# B&R Automation Studio project ABC_Pltzr (part 4)

### paiUDPService.typ - Global data types
```iecst
(********************************************************************
 * COPYRIGHT -- pai
 ********************************************************************
 * Package: paiUDPService
 * File: paiUDPService.typ
 * Author: goran
 * Created: October 12, 2011
 ********************************************************************
 * Data types of package paiUDPService
 ********************************************************************)

TYPE
	paiUdpConst_typ :
		(
		UDP_IP_ADDR_LEN := 32,
		UDP_SERVER_RXBUF_SIZE := 10000,
		UDP_CLIENT_TXBUF_SIZE := 10000
		);
	paiUdpIPAddress_typ : 	STRUCT
		digit3 : USINT;
		digit2 : USINT;
		digit1 : USINT;
		digit0 : USINT;
		text : STRING[20];
	END_STRUCT;
	paiUdpSystemConfig_typ : 	STRUCT
		magicNumber : UDINT; (*Magic number to detect permanent memory changes.*)
		udpClientMode : USINT; (*Outgoing (client) UDP mode of operation. 0-Echo (send status upon receiving command, needs only port number, used IP from received command), 1-Continues (needs host IP address and Port number)*)
		udpClientUpdateRate : USINT; (*Update rate (Hz) for the the UDP client when in mode 1;*)
		udpLocalServerPortNumber : UINT; (*UDP port number of the local UDP server.*)
		udpRemoteHostPortNumber : UINT; (*UDP port number of the remote host*)
		udpRemoteHostIpAddress : paiUdpIPAddress_typ; (*IP address of the remote UDP host*)
		updInterfaceType : UDINT; (*0-ISM native type; 1-Custom interface, type 1*)
	END_STRUCT;
	paiUdpStatistics_typ : 	STRUCT  (*UDP server statistics*)
		datagramCountTotal : UDINT; (*total number of received datagrams*)
		datagramPerSec : UDINT; (*number of received datagrams in the past second*)
		datagramPerSecMax : UDINT; (*max number of received datagrams in a second*)
		bytesTotal : UDINT; (*totral number of received bytes*)
		bytesPerSec : UDINT;
		bytesPerSecMax : UDINT;
		errorCountTotal : UDINT; (*total number of errors*)
	END_STRUCT;
	paiUdpClientInterface_typ : 	STRUCT
		iConnect : BOOL;
		iRmtIPAddr : STRING[UDP_IP_ADDR_LEN];
		iRmtUdpPort : UINT;
		iMode : USINT; (*0-echo mode (client's tx triggered by server's rx); 1-continues mode (rate timer 1 .. 100Hz used to trigger client's send) *)
		iSend : BOOL;
		iSendEcho : BOOL;
		iSendEchoRmtIpAddr : STRING[UDP_IP_ADDR_LEN];
		iUpdateRate : USINT;
		iTaskCycleTimeXms : USINT;
		iTxDataAdr : UDINT;
		iTxDataLen : UDINT;
		iTxCallback : UDINT;
		oError : BOOL;
		oRmtIpAddr : STRING[UDP_IP_ADDR_LEN];
		oRmtUdpPort : UINT;
		oConnected : BOOL;
		oSendDone : BOOL;
	END_STRUCT;
	paiUdpServerInterface_typ : 	STRUCT
		iEnable : BOOL;
		iUdpServerPort : UINT;
		iRxCallback : UDINT;
		iRxTimeoutXms : UDINT;
		oRxIsTimeout : BOOL;
		oError : BOOL;
		oRxReady : BOOL;
		oRxRmtIP : STRING[UDP_IP_ADDR_LEN];
		oRxRmtPort : UINT;
		oRxDataLen : UDINT;
		oRxDataLenMax : UDINT;
		oRxDataAdr : UDINT;
	END_STRUCT;
	paiUdpFBKs_typ : 	STRUCT
		open : UdpOpen;
		close : UdpClose;
		connect : UdpConnect;
		disconnect : UdpDisconnect;
		recv : UdpRecv;
		send : UdpSend;
		ioctl : UdpIoctl;
	END_STRUCT;
	paiUdpClient_typ : 	STRUCT
		clientIf : paiUdpClientInterface_typ;
		client : paiUdpFBKs_typ;
		txStats : paiUdpStatistics_typ;
		sm : bgSSM_typ;
		txbuf : ARRAY[0..UDP_CLIENT_TXBUF_SIZE]OF USINT;
	END_STRUCT;
	paiUdpServer_typ : 	STRUCT
		serverIf : paiUdpServerInterface_typ;
		server : paiUdpFBKs_typ;
		rxStats : paiUdpStatistics_typ;
		sm : bgSSM_typ;
		rmtIPAddr : STRING[UDP_IP_ADDR_LEN];
		rxlen : UDINT;
		rxbuf : ARRAY[0..UDP_SERVER_RXBUF_SIZE]OF USINT;
	END_STRUCT;
END_TYPE
```

### paiUDPService.var - Global variables
```iecst
(********************************************************************
 * COPYRIGHT -- pai
 ********************************************************************
 * Package: paiUDPService
 * File: paiUDPService.var
 * Author: goran
 * Created: October 12, 2011
 ********************************************************************
 * Variables of package paiUDPService
 ********************************************************************)
VAR CONSTANT
	gUdpServer_DefaultPort : UDINT := 9999; (*UDP Server default port*)
	gUdpClient_TaskCycleTimeXms : UDINT := 1; (*UDP Client task cycle time in [ms]*)
	gUdpClient_DefaultPort : UDINT := 9998; (*UDP Client default port*)
END_VAR
VAR
	gUdpClient_DefaultHostAdr : STRING[UDP_IP_ADDR_LEN] := '127.0.0.1'; (*UDP Client default host IP address when using continues UDP client mode*)
END_VAR
VAR RETAIN
	gUdpSystemCfg : paiUdpSystemConfig_typ := (0); (*UDP System Configuration Data (remanent memory)*)
END_VAR
VAR
	gUdpServer : paiUdpServer_typ; (*UDP Server Object Instance*)
	gUdpClient : paiUdpClient_typ; (*UDP Client Object Instance*)
END_VAR
```

### paiUdpserv.c - Implementation code
```c
/********************************************************************
 * COPYRIGHT -- pai
 ********************************************************************
 * Program: udpserv
 * File: udpserv.c
 * Author: goran
 * Created: October 05, 2011
 ********************************************************************
 * Implementation of program udpserv
 ********************************************************************/

#include <bur/plctypes.h>

#ifdef _DEFAULT_INCLUDES
	#include <AsDefault.h>
#endif

#include "../../libraries/sprintf2/sprintf2.h"

enum{
	udpServZero = 0,
	udpServEnable,
	udpServInit,
	udpServActive,
	udpServClose,
	udpServError,
	udpServLast
}STATEMACHINE;

static const char* udpServStateName(int state)
{
static const char* stateNames[] = {
"Zero",
"Enable",
"Init",
"Active",
"Close",
"Error",
};

	if( state >= udpServLast)
		return "unknow";

	return stateNames[state];
};

/*
###############################################################################
Utilities
###############################################################################
*/

/**
 Simple logging
 Log goes to an array of PV strings > see _LOCAL STRING log[][] variable below
 Log output is visible via Automation Studio watch window
 Example of a log statement used within the code is:
 DBG(lgr, "This is log example. %d ", value1);
 To complety disable logging from this source file, change next line to: #if 0
*/
#if 1
#include <../../bglib/bgPVLogger3.c>
#define LOG_ENTRY_COUNT 20	//max number of log entries
#define LOG_ENTRY_LENGTH  32 //max length of individual log message. Longer msg are truncated
_LOCAL STRING logUdpServ[LOG_ENTRY_COUNT][LOG_ENTRY_LENGTH]; //log output visible from Automation Studio!
#else
#define DBG(lgr, format, args...) ;
#define DBGINIT(lgr, logoutput, logEntryCount, logEntrySize)  ;
#endif

static void udpServerRxData(paiUdpServer_typ *p){
bgSSM_typ* pSm = &p->sm;

	//stats
	p->rxStats.datagramCountTotal++;
	p->rxStats.bytesTotal += p->server.recv.recvlen;

	//values for cummulative (per min) calculations
	pSm->counter[0]++;
	pSm->counter[1] +=p->server.recv.recvlen;

	//interface
	p->serverIf.oRxReady = 1;
	p->serverIf.oRxDataLen = p->server.recv.recvlen;
	p->serverIf.oRxDataAdr = (UDINT)p->rxbuf;
	p->serverIf.oRxRmtPort = p->server.recv.port;
	brsstrcpy((UDINT)p->serverIf.oRxRmtIP, (UDINT)p->rmtIPAddr);

	//execute rx callback to enable app to process received data
	if(p->serverIf.iRxCallback){
		void (*rxCallback)(UDINT pBuf, UDINT rxLen) =  ( void(*) (UDINT, UDINT) ) p->serverIf.iRxCallback;
		(*rxCallback)( (UDINT)p->rxbuf, p->server.recv.recvlen);
	}
}

/*
###############################################################################
Functions
###############################################################################
*/

static void udpServerSMCyclic(paiUdpServer_typ *p)
{
bgSSM_typ* pSm = &p->sm;

	//operate timer(s)
	bgTimerCyclic(&pSm->timer_x1ms[0]);
	bgTimerCyclic(&pSm->timer_x1ms[1]);//rx timeout timer
	bgTimerCyclic(&pSm->timer_x1ms[2]);//1 sec tick timer

	p->serverIf.oRxIsTimeout = bgTimerIsTimeOut(&pSm->timer_x1ms[1]);

	//stats timers
	if( bgTimerIsTimeOut(&pSm->timer_x1ms[2]) ){
		bgTimerStart(&pSm->timer_x1ms[2], 1000);

		//values for cummulative (per min) calculations for datagrams
		p->rxStats.datagramPerSec = pSm->counter[0];
		pSm->counter[0] = 0;
		if(p->rxStats.datagramPerSec > p->rxStats.datagramPerSecMax){
			p->rxStats.datagramPerSecMax = p->rxStats.datagramPerSec;
		}

		//values for cummulative (per min) calculations for bytes
		p->rxStats.bytesPerSec = pSm->counter[1];
		pSm->counter[1] = 0;
		if(p->rxStats.bytesPerSec > p->rxStats.bytesPerSecMax){
			p->rxStats.bytesPerSecMax = p->rxStats.bytesPerSec;
		}
	}

	/*execute control state machine cyclic handler*/
	bgSSMCyclic(pSm);
	//show change of state in a log
	if( bgSSMIsStateInit(pSm) ){
		DBG(lgr, "sm=%s(%d)", bgSSMGetStateText(pSm), bgSSMGetState(pSm));
	}

	switch(bgSSMGetState(pSm)){
		//========================================
		case udpServZero:
			bgSSMStateNext(pSm, udpServEnable);
			p->serverIf.oError = 0;
			p->serverIf.oRxReady = 0;

		break;
		//========================================
		case udpServEnable:
			if(p->serverIf.iEnable){
				bgSSMStateNext(pSm, udpServInit);
			}
		break;
		//========================================
		case udpServInit:

			if( bgSSMIsStateInit(pSm) ){

				p->server.open.enable = 1;
				p->server.open.port = p->serverIf.iUdpServerPort;
				p->server.open.pIfAddr = 0;
//IMPORTANT:
//in order for the following conditional compilation to work properly, PLC object in the Configuration view
//must contain following defintion:
//Folder: Build
//Field: Additional Build Options
//Value: -D $(AS_CONFIGURATION)
//Using the above, name of the current AS configuration (i.e. realhw1 or testsim or else) becomes
//a defined preprocessor name. As a result, it's possible to destinguish between different configurations!
//#ifdef testsim
#ifdef Simulation
				//In case of testsim (ARsim) target, don't use socket options
				p->server.open.options = 0;
#warning "Project - UDP - ARsim target!"
#else
				//For all other (real) targets, use socket options
				p->server.open.options = udpOPT_REUSEPORT;
#warning "Project - UDP - NOT an ARsim target!"
#endif
				return;
			}

			if(p->server.open.status == ERR_FUB_BUSY)
				return;

			p->server.open.enable = 0;

			if(p->server.open.status == ERR_OK){
				p->server.recv.ident = p->server.open.ident;
				p->server.send.ident = p->server.open.ident;
				p->server.close.ident = p->server.open.ident;
				p->server.connect.ident = p->server.open.ident;
				p->server.disconnect.ident = p->server.open.ident;
				p->server.ioctl.ident = p->server.open.ident;
				bgSSMStateNext(pSm, udpServActive);
				return;
			}

			DBG(lgr,"Err udp.open=%d", p->server.open.status);
			bgSSMStateNext(pSm, udpServError);

		break;
		//========================================
		case udpServActive:

			if( bgSSMIsStateInit(pSm) ){
				p->server.recv.enable = 1;

				p->server.recv.pData = (UDINT)&p->rxbuf[0];
				p->server.recv.datamax = UDP_SERVER_RXBUF_SIZE;
				p->server.recv.pIpAddr = (UDINT)&p->rmtIPAddr[0];
				p->server.recv.flags = 0;

				bgTimerStart(&pSm->timer_x1ms[1], p->serverIf.iRxTimeoutXms);

				return;
			}

			//Disabling UDP server currently not supported. Disabling (i.e. change port) requires reset
			//if(!p->serverIf.iEnable){
			//	stateNext(pSm, udpServClose);
			//}

			if((p->server.recv.status == ERR_FUB_BUSY) || (p->server.recv.status == udpERR_NO_DATA))
				return;

			p->server.recv.enable = 0;

			if(p->server.recv.status == ERR_OK){

				DBG(lgr,"udpServ rx from %s", p->rmtIPAddr);
				DBG(lgr,"rmtPort=%d, rxlen=%d", p->server.recv.port, p->server.recv.recvlen);
				udpServerRxData(p);
				return;
			}

			DBG(lgr,"Err udp.recv=%d", p->server.recv.status);
			bgSSMStateNext(pSm, udpServError);

		break;
		//========================================
		case udpServClose:

			if( bgSSMIsStateInit(pSm) ){
				DBG(lgr,"UDP Server close");
				p->server.close.enable = 1;
				p->server.recv.enable = 0;
				return;
			}

			if(p->server.close.status == ERR_FUB_BUSY)
				return;

			if(p->server.close.status){
				DBG(lgr,"Err udp.close=%d", p->server.close.status);
			}

			p->server.close.enable = 0;

			bgSSMStateNext(pSm, udpServZero);
		break;
		//========================================
		case udpServError:

			if( bgSSMIsStateInit(pSm) ){
				DBG(lgr,"UDP Server Error State");

				//start error recovery timer
				bgTimerStart(&pSm->timer_x1ms[0], 5000);
			}

			if( bgTimerIsTimeOut(&pSm->timer_x1ms[0]) ){
				//after timer exp > try to close the port and see if it recovers
				bgSSMStateNext(pSm, udpServClose);
			}

		break;
		//========================================
		default:
		break;
	}

}

static void udpServerInit(paiUdpServer_typ *p)
{
	bgSSM_typ* pSm = &p->sm;

	brsmemset((UDINT)p, 0, sizeof(paiUdpServer_typ));

	bgTimerStart(&p->sm.timer_x1ms[2], 1000);

	bgSSMInit(pSm, (UDINT)udpServStateName, 0);
}

static void udpServerCyclic(paiUdpServer_typ *p)
{
	//udp server state machine cyclic
	udpServerSMCyclic(p);

	//udp server fbk-s
	UdpOpen(&p->server.open);
	UdpClose(&p->server.close);
	UdpConnect(&p->server.connect);
	UdpDisconnect(&p->server.disconnect);
	UdpSend(&p->server.send);
	UdpRecv(&p->server.recv);
	UdpIoctl(&p->server.ioctl);

}

/*
###############################################################################
Main entry: Init & Cyclic Functions
###############################################################################
*/
void paiUdpServerInit(paiUdpServer_typ *p)
{
	/* TODO: Add code here */

	//init logger object
	DBGINIT(lgr, logUdpServ, LOG_ENTRY_COUNT, LOG_ENTRY_LENGTH);
	DBG(lgr, "INIT: paiUdpServerInit");

	//udp server init
	udpServerInit(p);

}

void paiUdpServerCyclic(paiUdpServer_typ *p)
{
	/* TODO: Add code here */
	//udp server cyclic
	udpServerCyclic(p);
}
```

### paiUdpclient.c - Implementation code
```c
/********************************************************************
 * COPYRIGHT -- pai
 ********************************************************************
 * Program: udpclient
 * File: udpclient.c
 * Author: goran
 * Created: January 23, 2013
 ********************************************************************
 * Implementation of program udpclient
 ********************************************************************/

#include <bur/plctypes.h>

#ifdef _DEFAULT_INCLUDES
	#include <AsDefault.h>
#endif

#include <../../bglib/bgstring.h>
#include "../../libraries/sprintf2/sprintf2.h"

enum{
	udpCliZero = 0,
	udpCliInit,
	udpCliOpen,
	udpCliConnect,
	udpCliIdle,
	udpCliTxData,
	udpCliDisconnect,
	udpCliClose,
	udpCliError,
	udpCliLast
}STATEMACHINE;

static const char* udpCliStateName(int state)
{
static const char* stateNames[] = {
"Zero",
"Init",
"Open",
"Connect",
"Idle",
"TxData",
"Disconnect",
"Close",
"Error",
};

	if( state >= udpCliLast)
		return "unknow";

	return stateNames[state];
};

/*
###############################################################################
Utilities
###############################################################################
*/

static void convertIPTextToDigits(paiUdpIPAddress_typ* p)
{
unsigned char txtbuffer[64];
bgStringList_typ list;

	brsstrcpy((UDINT)txtbuffer, (UDINT)(p->text));
	list.src = txtbuffer;

	bgStringSplitLine(&list, '.');
	if(list.itemCount != 4){
		p->digit3 = 0;
		p->digit2 = 0;
		p->digit1 = 0;
		p->digit0 = 0;
		return;
	}
	p->digit3 = (USINT)brsatoi((UDINT)list.items[0]);
	p->digit2 = (USINT)brsatoi((UDINT)list.items[1]);
	p->digit1 = (USINT)brsatoi((UDINT)list.items[2]);
	p->digit0 = (USINT)brsatoi((UDINT)list.items[3]);
}

/**
 Simple logging
 Log goes to an array of PV strings > see _LOCAL STRING log[][] variable below
 Log output is visible via Automation Studio watch window
 Example of a log statement used within the code is:
 DBG(lgr, "This is log example. %d ", value1);
 To complety disable logging from this source file, change next line to: #if 0
*/
#if 1
#include <../../bglib/bgPVLogger3.c>
#define LOG_ENTRY_COUNT 20	//max number of log entries
#define LOG_ENTRY_LENGTH  32 //max length of individual log message. Longer msg are truncated
_LOCAL STRING logUdpClient[LOG_ENTRY_COUNT][LOG_ENTRY_LENGTH]; //log output visible from Automation Studio!
#else
#define DBG(lgr, format, args...) ;
#define DBGINIT(lgr, logoutput, logEntryCount, logEntrySize)  ;
#endif

/*
###############################################################################
Functions
###############################################################################
*/

static void udpClientSMCyclic(paiUdpClient_typ *p)
{
bgSSM_typ* pSm = &p->sm;

	//operate timer(s)
	bgTimerCyclic(&pSm->timer_x1ms[0]); // delay timer

	//TimerExecute(&pSm->timer2x1ms); // update rate timer (in continues mode)
	//IMPORANT: for high speed, can't use TON block > rather, use cycle time
	if(pSm->timer_x1ms[1].ET)
		pSm->timer_x1ms[1].ET--;

	bgTimerCyclic(&pSm->timer_x1ms[2]); // 1sec stats timer

	//stats timers
	if( bgTimerIsTimeOut(&pSm->timer_x1ms[2]) ){
		bgTimerStart(&pSm->timer_x1ms[2], 1000);

		//values for cummulative (per min) calculations for datagrams
		p->txStats.datagramPerSec = pSm->counter[0];
		pSm->counter[0] = 0;
		if(p->txStats.datagramPerSec > p->txStats.datagramPerSecMax){
			p->txStats.datagramPerSecMax = p->txStats.datagramPerSec;
		}

		//values for cummulative (per min) calculations for bytes
		p->txStats.bytesPerSec = pSm->counter[1];
		pSm->counter[1] = 0;
		if(p->txStats.bytesPerSec > p->txStats.bytesPerSecMax){
			p->txStats.bytesPerSecMax = p->txStats.bytesPerSec;
		}
	}

	/*execute control state machine cyclic handler*/
	bgSSMCyclic(pSm);

	//show change of state in a log
	if( bgSSMIsStateInit(pSm) ){
		DBG(lgr, "sm=%s(%d)", bgSSMGetStateText(pSm), bgSSMGetState(pSm));
	}

	switch( bgSSMGetState(pSm) ){
		//========================================
		case udpCliZero:
			bgSSMStateNext(pSm, udpCliInit);
		break;
		//========================================
		case udpCliInit:
			if(p->clientIf.iConnect){
				bgSSMStateNext(pSm, udpCliOpen);
			}
		break;
		//========================================
		case udpCliOpen:

			if( bgSSMIsStateInit(pSm) ){
				p->client.open.enable = 1;
				p->client.open.port = 0;
				p->client.open.pIfAddr = 0;
//IMPORTANT:
//in order for the following conditional compilation to work properly, PLC object in the Configuration view
//must contain following defintion:
//Folder: Build
//Field: Additional Build Options
//Value: -D $(AS_CONFIGURATION)
//Using the above, name of the current AS configuration (i.e. realhw1 or testsim or else) becomes
//a defined preprocessor name. As a result, it's possible to destinguish between different configurations!
//#ifdef testsim
#ifdef Simulation
				//In case of testsim (ARsim) target, don't use socket options
				p->client.open.options = 0;
#warning "UDP Client - ARsim target!"
#else
				//For all other (real) targets, use socket options
				p->client.open.options = udpOPT_REUSEPORT | udpOPT_BROADCAST;
#warning "UDP Client - real target!"
#endif
				return;
			}

			if(p->client.open.status == ERR_FUB_BUSY)
				return;

			p->client.open.enable = 0;

			if(p->client.open.status == ERR_OK){
				p->client.recv.ident = p->client.open.ident;
				p->client.send.ident = p->client.open.ident;
				p->client.close.ident = p->client.open.ident;
				p->client.connect.ident = p->client.open.ident;
				p->client.disconnect.ident = p->client.open.ident;
				p->client.ioctl.ident = p->client.open.ident;
				bgSSMStateNext(pSm, udpCliConnect);
				return;
			}

			DBG(lgr,"Err udp.open=%d", p->client.open.status);
			bgSSMStateNext(pSm, udpCliError);

		break;
		//========================================
		case udpCliConnect:

			if( bgSSMIsStateInit(pSm) ){
				p->client.connect.enable = 1;
				p->client.connect.port = p->clientIf.iRmtUdpPort;
				p->client.connect.pHost = (UDINT)p->clientIf.iRmtIPAddr;
				return;
			}

			if(p->client.connect.status == ERR_FUB_BUSY)
				return;

			//p->client.connect.enable = 0;

			if(p->client.connect.status == ERR_OK){
				brsstrcpy((UDINT)p->clientIf.oRmtIpAddr, (UDINT)p->clientIf.iRmtIPAddr);
				p->clientIf.oRmtUdpPort = p->clientIf.iRmtUdpPort;

				bgSSMStateNext(pSm, udpCliIdle);
				return;
			}

			DBG(lgr,"Err udp.connect=%d", p->client.connect.status);
			bgSSMStateNext(pSm, udpCliError);

		break;
		//========================================
		case udpCliIdle:

			if( bgSSMIsStateInit(pSm) ){

			}

			//udp client in echo mode!?
			//check for iSendEcho set by the server upon it receives a message > client sends out to the same host
			if(!p->clientIf.iMode && p->clientIf.iSendEcho){
				p->clientIf.iSendEcho = 0;
				p->clientIf.iSend = 1;
				brsstrcpy((UDINT)p->clientIf.iRmtIPAddr, (UDINT)p->clientIf.iSendEchoRmtIpAddr);
			}

			//udp client in continues mode!?
			//trigger send update at a configured rate to a defined (sipplied to the inputs) remote host/port
			if(p->clientIf.iMode){

				if(!pSm->timer_x1ms[1].ET){
					int updateTimeMs;

					if( p->clientIf.iUpdateRate ){
						updateTimeMs = 1000 /  p->clientIf.iUpdateRate;
					}else{
						updateTimeMs = 1000;
					}

					if(updateTimeMs < 10)
						updateTimeMs = 12;

					if(updateTimeMs > 1000)
						updateTimeMs = 1000;

					if(p->clientIf.iTaskCycleTimeXms){
						pSm->timer_x1ms[1].ET= updateTimeMs / p->clientIf.iTaskCycleTimeXms;
					}else{
						pSm->timer_x1ms[1].ET= updateTimeMs / gUdpClient_TaskCycleTimeXms; // devide by task clas time to find out increments
					}

					p->clientIf.iSend = 1;
				}

			}

			//monitor for change in remote host settings
			//in case of a change > reconnect (disconncet then connect)
			if((p->clientIf.oRmtUdpPort != p->clientIf.iRmtUdpPort) ||
				brsstrcmp((UDINT)p->clientIf.oRmtIpAddr, (UDINT)p->clientIf.iRmtIPAddr)
			){
				DBG(lgr,"rmt settings changed. Triggering reconnect.");
				bgSSMStateNext(pSm, udpCliDisconnect);
				return;
			}

			//monitor request to send
			if(p->clientIf.iSend){
				p->clientIf.iSend = 0;

				if(p->clientIf.iTxDataLen > UDP_CLIENT_TXBUF_SIZE){
					p->clientIf.iTxDataLen = UDP_CLIENT_TXBUF_SIZE;
				}

				if(!p->clientIf.iTxDataAdr && !p->clientIf.iTxCallback){
					DBG(lgr,"udp.send nothing to tx");
					return;
				}

				//execute memcpy if datasource is defined
				if(p->clientIf.iTxDataAdr){
					brsmemcpy((UDINT)(p->txbuf), (UDINT)(p->clientIf.iTxDataAdr), p->clientIf.iTxDataLen);
				}

				//execute callback to enable app to populate data before sending
				//NOTE: callback will overwrite effect of the above memcpy if both a defined!!!
				if(p->clientIf.iTxCallback){
					void (*txCallback)(UDINT pBuf, UDINT lenTxBuf, UDINT* pLenData) =  ( void(*) (UDINT, UDINT, UDINT*) ) p->clientIf.iTxCallback;
					(*txCallback)( (UDINT)&p->txbuf[0], UDP_CLIENT_TXBUF_SIZE, &p->clientIf.iTxDataLen);
				}

				p->client.send.enable = 1;
				p->client.send.pData = (UDINT)&p->txbuf[0];
				p->client.send.datalen = p->clientIf.iTxDataLen;

				//stats
				p->txStats.datagramCountTotal++;
				p->txStats.bytesTotal += p->client.send.datalen;

				//values for cummulative (per min) calculations
				pSm->counter[0]++;
				pSm->counter[1] +=p->client.send.datalen;

				bgSSMStateNext(pSm, udpCliTxData);
				return;
			}

		break;
		//========================================
		case udpCliTxData:
			if( bgSSMIsStateInit(pSm) ){

			}

			if(p->client.send.status == ERR_FUB_BUSY)
				return;

			p->client.send.enable = 0;

			if(p->client.send.status == ERR_OK){
				p->clientIf.oSendDone = 1;
				DBG(lgr,"udp.send OK");
				bgSSMStateNext(pSm, udpCliIdle);
				return;
			}

			DBG(lgr,"Err udp.send=%d", p->client.send.status);
			bgSSMStateNext(pSm, udpCliError);

		break;
		//========================================
		case udpCliDisconnect:

			if( bgSSMIsStateInit(pSm) ){
				p->client.connect.enable = 0;
				p->client.disconnect.enable = 1;
				return;
			}

			if(p->client.disconnect.status == ERR_FUB_BUSY)
				return;

			p->client.disconnect.enable = 0;

			if(p->client.disconnect.status == ERR_OK){
				bgSSMStateNext(pSm, udpCliClose);
				return;
			}

			DBG(lgr,"Err udp.disconnect=%d", p->client.disconnect.status);
			bgSSMStateNext(pSm, udpCliClose);

		break;
		//========================================
		case udpCliClose:

			if( bgSSMIsStateInit(pSm) ){
				DBG(lgr,"UDP Client close");
				p->client.close.enable = 1;
				return;
			}

			if(p->client.close.status == ERR_FUB_BUSY)
				return;

			if(p->client.close.status){
				DBG(lgr,"Err udp.close=%d", p->client.close.status);
			}

			p->client.close.enable = 0;

			bgSSMStateNext(pSm, udpCliZero);
		break;
		//========================================
		case udpCliError:

			if( bgSSMIsStateInit(pSm) ){
				DBG(lgr,"UDP Client Error State");

				//start error recovery timer
				bgTimerStart(&pSm->timer_x1ms[0], 5000);
			}

			if( bgTimerIsTimeOut(&pSm->timer_x1ms[0]) ){
				//after timer exp > try to close the port and see if it recovers
				bgSSMStateNext(pSm, udpCliDisconnect);
			}

		break;
		//========================================
		default:
		break;
	}

}

void udpClientInit(paiUdpClient_typ *p)
{
	bgSSM_typ* pSm = &p->sm;

	bgTimerStart(&p->sm.timer_x1ms[2], 1000);

	bgSSMInit(pSm, (UDINT)udpCliStateName, 0);

}

void udpClientCyclic(paiUdpClient_typ *p)
{

	//udp client state machine
	udpClientSMCyclic(p);

	//udp client fbk-s
	UdpOpen(&p->client.open);
	UdpClose(&p->client.close);
	UdpConnect(&p->client.connect);
	UdpDisconnect(&p->client.disconnect);
	UdpSend(&p->client.send);
	UdpRecv(&p->client.recv);
	UdpIoctl(&p->client.ioctl);
}
/*
###############################################################################
Main entry: Init & Cyclic Functions
###############################################################################
*/

void paiUdpClientInit(paiUdpClient_typ *p)
{
	/* TODO: Add code here */

	//init logger object
	DBGINIT(lgr, logUdpClient, LOG_ENTRY_COUNT, LOG_ENTRY_LENGTH);
	DBG(lgr, "INIT: paiUdpClientInit");

	udpClientInit(p);

	//upd client application specific init
	p->clientIf.iConnect = 1;
#if 0

	//RESTORE SETTINGS FROM THE REMANENT STORAGE
	//sanity check for remote host ip address
	convertIPTextToDigits(&gUdpSystemCfg.udpRemoteHostIpAddress);

	if(!gUdpSystemCfg.udpRemoteHostIpAddress.digit0 ||
		!gUdpSystemCfg.udpRemoteHostIpAddress.digit1 ||
		!gUdpSystemCfg.udpRemoteHostIpAddress.digit2 ||
		!gUdpSystemCfg.udpRemoteHostIpAddress.digit3
	){
		brsstrcpy((UDINT)gUdpSystemCfg.udpRemoteHostIpAddress.text, (UDINT)gUdpClient_DefaultHostAdr);
		convertIPTextToDigits(&gUdpSystemCfg.udpRemoteHostIpAddress);
	}
	brsstrcpy((UDINT)gUdpClient.clientIf.iRmtIPAddr, (UDINT)gUdpSystemCfg.udpRemoteHostIpAddress.text);

	//sanity check for remote host UDP port number
	if(!gUdpSystemCfg.udpRemoteHostPortNumber){
		gUdpSystemCfg.udpRemoteHostPortNumber = gUdpClient_DefaultPort;
	}
	gUdpClient.clientIf.iRmtUdpPort = gUdpSystemCfg.udpRemoteHostPortNumber;

	// udpClientMode
	// 0-echo mode (send status after receiving a command from the host. Uses received IP address and UDP port number configured here.
	// 1-continues mode (send status independantly to configured 	remoteIpAddress. remoteUDP port at the configure UDP rate
	if(gUdpSystemCfg.udpClientMode > 1){
		gUdpSystemCfg.udpClientMode = 0;
	}
	gUdpClient.clientIf.iMode = gUdpSystemCfg.udpClientMode;

	// udpClientUpdateRate
	// rate to send outgoing status to remote host in case of UDP client mode 1
	//
	if(gUdpSystemCfg.udpClientUpdateRate < 1){
		gUdpSystemCfg.udpClientUpdateRate  = 1;
	}
	if(gUdpSystemCfg.udpClientUpdateRate > 100){
		gUdpSystemCfg.udpClientUpdateRate  = 100;
	}
	gUdpClient.clientIf.iUpdateRate = gUdpSystemCfg.udpClientUpdateRate;

	gUdpClient.clientIf.iSend = 0;

#endif
	//dgsUdpClientInit();
}

void  paiUdpClientCyclic(paiUdpClient_typ *p)
{
	/* TODO: Add code here */

	//udp client cyclic
	udpClientCyclic(p);

#if 0
	//in continues client mode, use localy configured settings!
	if(/*gUdpSystemCfg.udpClientMode &&*/
		((gUdpSystemCfg.udpClientMode != gUdpClient.clientIf.iMode) ||
		(gUdpClient.clientIf.iUpdateRate != gUdpSystemCfg.udpClientUpdateRate) ||
		brsstrcmp((UDINT)gUdpClient.clientIf.iRmtIPAddr, (UDINT)gUdpSystemCfg.udpRemoteHostIpAddress.text))
	){
		gUdpClient.clientIf.iMode = gUdpSystemCfg.udpClientMode;
		gUdpClient.clientIf.iUpdateRate = gUdpSystemCfg.udpClientUpdateRate;
 		brsstrcpy((UDINT)gUdpClient.clientIf.iRmtIPAddr, (UDINT)gUdpSystemCfg.udpRemoteHostIpAddress.text);
	}

	//in echo mode, just monitor for iMode change
	if(!gUdpSystemCfg.udpClientMode &&
		((gUdpSystemCfg.udpClientMode != gUdpClient.clientIf.iMode) )
	){
		gUdpClient.clientIf.iMode = gUdpSystemCfg.udpClientMode;
	}

	//in both modes use configured port number for the remote UDP host
	gUdpClient.clientIf.iRmtUdpPort = gUdpSystemCfg.udpRemoteHostPortNumber;

	//udp client cyclic
	//dgsUdpClientCyclic();
#endif
}
```

### paiUdpService.h
```c
/********************************************************************
 * COPYRIGHT --
 ********************************************************************
 * Package: paiUDPService
 * File: paiUdpService.h
 * Author: goran
 * Created: June 22, 2015
 *******************************************************************/

#include <bur/plctypes.h>

#ifdef _DEFAULT_INCLUDES
	#include <AsDefault.h>
#endif

void paiUdpServerInit(paiUdpServer_typ *p);
void paiUdpServerCyclic(paiUdpServer_typ *p);
void paiUdpClientInit(paiUdpClient_typ *p);
void paiUdpClientCyclic(paiUdpClient_typ *p);
```

### Program Logical/paiComponents/paiUDP/udpApp

#### udpApp.c
```c
/********************************************************************
 * COPYRIGHT -- pai
 ********************************************************************
 * Program: appUDP
 * File: appUDP.c
 * Author: goran
 * Created: Jan 25, 2013
 ********************************************************************
 * Implementation of program appUDP
 ********************************************************************/

#include <bur/plctypes.h>

#ifdef _DEFAULT_INCLUDES
	#include <AsDefault.h>
#endif

#include <../../../libraries/sscanf2/sscanf2.h>
#include <../paiUdpService/paiUdpService.h>
#include "../../libraries/sprintf2/sprintf2.h"
#include "../../libraries/bgringbuf/bgringbuffer.h"

#include <../../../ProjGlob/ipc.h>
#include "../../../ProjGlob/GlobalDec.h"

/*
###############################################################################
Utilities
###############################################################################
*/

/**
 Simple logging
 Log goes to an array of PV strings > see _LOCAL STRING log[][] variable below
 Log output is visible via Automation Studio watch window
 Example of a log statement used within the code is:
 DBG(lgr, "This is log example. %d ", value1);
 To complety disable logging from this source file, change next line to: #if 0
IMPORTANT:
==========
DBGINIT() statement MUST BE PLACED as a first statement within the task _INIT function!
Example:
void _INIT myTaskINIT(void)
{
	//TODO: Add code here
	//init logger object
	DBGINIT(lgr, log, LOG_ENTRY_COUNT, LOG_ENTRY_LENGTH);
}
*/
#if 1
#include <../../bglib/bgPVLogger3.c>
#define LOG_ENTRY_COUNT 100	//max number of log entries
#define LOG_ENTRY_LENGTH  100 //max length of individual log message. Longer msg are truncated
_LOCAL STRING logUdpApp[LOG_ENTRY_COUNT][LOG_ENTRY_LENGTH]; //log output visible from Automation Studio!
#else
#define DBG(lgr, format, args...) ;
#define DBGINIT(lgr, logoutput, logEntryCount, logEntrySize)  ;
#endif

/**
###############################################################################
UDP Server Receive function
###############################################################################
*/
static void udpServerCallback(UDINT pRxBuffer, UDINT lenRxData)
{

	DBG(lgr, "udpServerCallback lenRxData=%d\n\r", lenRxData);
}

/**
###############################################################################
UDP callback functions
###############################################################################
*/
//UDP Server Receive function
static void udpServerCallbackAfterReceive(UDINT pRxBuffer, UDINT lenRxData)
{
	udpServerCallback(pRxBuffer, lenRxData);
}

//UDP Client Send Callback function
static void udpClientCallback(UDINT pTxBuffer, UDINT lenTxBuffer, UDINT* pTxDataLen)
{
//	(*pTxDataLen) = brsstrlen((UDINT)&gUdpClient.txbuf[0]);
}

//UDP Client Send Callback function
static void udpClientCallbackBeforeSend(UDINT pTxBuffer, UDINT lenTxBuffer, UDINT* pTxDataLen)
{
	udpClientCallback(pTxBuffer, lenTxBuffer, pTxDataLen);
}

/*
###############################################################################
UDP communication timeout handler
###############################################################################
*/
static void	udpTimeOutHandler()
{
	//application logic - an example of handling a UDP receive timeout event
	//static BOOL oldRxTimeout;
	if( gUdpRxState && bgTimerIsTimeOut(&gUdpCommTimeoutTmr) /*&& !gYPAlarms.alarmActive[APP_ALARM_DBPROXYTIMEOUT]*/){
		DBG(lgr, "udp server rx timeout");
		//gYPAlarms.alarmActive[APP_ALARM_DBPROXYTIMEOUT] = gConfig.active.diag.disableDBProxTimeoutAlarm ? 0 : 1;
	}
}

/*
###############################################################################
Task execution entry points: Init & Cyclic Functions
###############################################################################
*/
void _INIT udpAppINIT(void)
{

	/* TODO: Add code here */
	//init logger object
	DBGINIT(lgr, logUdpApp, LOG_ENTRY_COUNT, LOG_ENTRY_LENGTH);
	DBG(lgr, "INIT: udpAppINIT");

	//Init UDP server object
	//======================
	paiUdpServerInit(&gUdpServer);
	//Set UDP server related parameters
	//Define application specific UDP server rx callback function
	gUdpServer.serverIf.iRxCallback = (UDINT)udpServerCallbackAfterReceive;
	gUdpServer.serverIf.oRxDataLenMax = UDP_SERVER_RXBUF_SIZE;
	gUdpServer.serverIf.iEnable = 1;
	gUdpServer.serverIf.iUdpServerPort = 9999;

	//Init UDP client object
	//======================
	paiUdpClientInit(&gUdpClient);

	//Define application specific UDP client tx callback function
	gUdpClient.clientIf.iTxCallback = (UDINT)udpClientCallbackBeforeSend;

	//Adjust UDP client/server settings according to the application needs (i.e. use HMI if needed)
	//For other defaults see:
	//paiUDPService.var (i.e. defined UDP related const)
	//udpserv.c/udpservINIT() and udpclient.c/udpclientINIT()
	gUdpSystemCfg.udpClientMode = 0;//not continues mode
	gUdpSystemCfg.udpClientUpdateRate = 10;//[Hz]
	//strcpy(gUdpSystemCfg.udpRemoteHostIpAddress.text, "192.168.100.31");
	//strcpy(gUdpSystemCfg.udpRemoteHostIpAddress.text, "192.168.100.171");
	brsstrcpy((UDINT)gUdpSystemCfg.udpRemoteHostIpAddress.text, (UDINT)"192.168.100.255");
	//strcpy(gUdpSystemCfg.udpRemoteHostIpAddress.text, "192.168.100.10");
	//strcpy(gUdpSystemCfg.udpRemoteHostIpAddress.text, "127.0.0.1");
	//strcpy(gUdpSystemCfg.udpRemoteHostIpAddress.text, "192.168.100.255");
	gUdpClient.clientIf.iTaskCycleTimeXms = 1;//udp client runs under 10ms cycle time
	gUdpServer.serverIf.iRxTimeoutXms = 4000;//udp server rx timeout time

	//bgTimerStart(&gUdpCommTimeoutTmr, gConfig.active.hmi.dbProxyCommTimeout * 1000.0);//start response timeout timer
	bgTimerStart(&gUdpCommTimeoutTmr, 5000);//start response timeout timer

}

//typedef union TAppIpcMsgXXX
//{
//    UDINT gen;
//    USINT rw_shm;
//    DINT  errMsg;
//}TAppIpcMsgXXX_typ;
//

void _CYCLIC udpAppCYCLIC(void)
{
	/* TODO: Add code here */

	//operate timer
	bgTimerCyclic(&gUdpCommTimeoutTmr) ;

	//application logic - on send complete, copy status into last statusSent
	if(gUdpClient.clientIf.oSendDone){
		gUdpClient.clientIf.oSendDone = 0;

		overheadIpcUDPTxClientCyclic( &gIpcCommFifoMem );

		//preset response timeout timer
//		gUdpRxState = 1; //need to receive a response
		if( bgTimerIsTimeOut(&gUdpCommTimeoutTmr) ){
			//bgTimerStart(&gUdpCommTimeoutTmr, gConfig.active.hmi.dbProxyCommTimeout * 1000.0);//start response timeout timer
			bgTimerStart(&gUdpCommTimeoutTmr, 5000);//start response timeout timer
		}
	}

	//application logic - en example of handling a UDP rx event
	if(gUdpServer.serverIf.oRxReady){
		//gUdpServer.serverIf.oRxReady = 0; //Consumer of the message shall clear this bit
		gUdpRxState = 0; //response received
		//gYPAlarms.alarmActive[APP_ALARM_DBPROXYTIMEOUT] = 0;//clear DB proxy alarm
	}

	//handle a UDP rx timeout
	udpTimeOutHandler();

	//cyclic execution of the UDP related services
	paiUdpServerCyclic(&gUdpServer);
	paiUdpClientCyclic(&gUdpClient);
}
//EOF
```

### paiUser.typ - pai Mp types
```iecst
(********************************************************************
 * COPYRIGHT -- pai
 ********************************************************************
 * Package: paiTemplate
 * File: paiUser.typ
 * Author: goran
 * Created: August 28, 2013
 ********************************************************************
 * Data types of package paiUser
 ********************************************************************)
(*########################################################################*)
(*pai specific defines for user access logic*)
(*########################################################################*)

TYPE
	paiUserAccessMaxEnums :
		(
		paiUSER_RIGHTSMAXIDX := 19, (*Access rights max index*)
		paiUSER_USERSMAXIDX := 9, (*Users max index*)
		paiUSER_GROUPMAXIDX := 5 (*Groups max index*)
		);
	paiUserAccessRightsIndex :
		(
		paiUSER_ACCESS_MFG := 0, (*Access right index*)
		paiUSER_ACCESS_ADMIN := 1, (*Access right index*)
		paiUSER_ACCESS_MAINT := 2, (*Access right index*)
		paiUSER_ACCESS_NONE := 3 (*Access right index*)
		);
	paiMpUserAccessRightEnum :
		(
		mpUSER_ACCESS_UNDEFINED := 0, (*Access right undefined*)
		mpUSER_ACCESS_NONE := 1, (*No access rights*)
		mpUSER_ACCESS_VIEW := 2, (*Read access*)
		mpUSER_ACCESS_ACTUATE := 3, (*Processes can be started/stopped but not edited*)
		mpUSER_ACCESS_FULL := 4 (*Full access (read-write access)*)
		);
	paiMpUserMgrUIGroupInfoType : 	STRUCT
		Name : STRING[20]; (*Name of the user group*)
		Index : UINT; (*Index of the user group*)
		Level : DINT; (*Level of the user group*)
		Admin : BOOL; (*Indicates whether this group has administrator rights*)
		AccessRights : ARRAY[0..19]OF paiMpUserAccessRightEnum; (*List with the access rights for individual actions*)
	END_STRUCT;
	paiUserInfo_typ : 	STRUCT
		UserName : STRING[20];
		UserFullName : STRING[100];
		Password : STRING[20];
		PIN : UDINT;
		GroupIndex : UDINT;
	END_STRUCT;
	paiUserMgrUIConnect_typ : 	STRUCT
		groupIndex : UDINT;
		groupIndexMax : UDINT;
		userIndex : UDINT;
		userIndexMax : UDINT;
		loggedIndex : UDINT;
		isUserLogged : UDINT;
		visibleLogged : UDINT;
		visibleNotLogged : UDINT;
		btnRestartLoginTimer : UDINT;
		btnToggleLogin : UDINT;
		remainingLoginTime_min : UDINT;
		remainingLoginTime_sec : UDINT;
		pwdLevel : UDINT;
		pwdLevelOld : UDINT;
		pwdLevelCompletion : UDINT;
		listUserNames : ARRAY[0..11]OF STRING[20];
		listUserPasswords : ARRAY[0..11]OF STRING[20];
	END_STRUCT;
	paiUserMgrPrivate_typ : 	STRUCT
		UIConnect : paiUserMgrUIConnect_typ;
		loginTimer : TON;
	END_STRUCT;
	paiUserConfiguration_typ : 	STRUCT
		listGroups : ARRAY[0..5]OF paiMpUserMgrUIGroupInfoType; (*table colum: id-s*)
		listUsers : ARRAY[0..9]OF paiUserInfo_typ;
		loginTime_sec : REAL;
		New_Member : USINT;
	END_STRUCT;
	paiUserMgr_typ : 	STRUCT
		currentGroup : paiMpUserMgrUIGroupInfoType;
		currentUser : paiUserInfo_typ;
		pUserConfig : REFERENCE TO paiUserConfiguration_typ;
		userMgr : paiUserMgrPrivate_typ;
	END_STRUCT;
END_TYPE
```

### paiUser.var - Global variables
```iecst
(********************************************************************
 * COPYRIGHT -- pai
 ********************************************************************
 * Package: HMI
 * File: HMI.var
 * Author: goran
 * Created: August 28, 2013
 ********************************************************************
 * Variables of package HMI
 ********************************************************************)
VAR
	gPaiUserConfig : paiUserConfiguration_typ := (0);
	gPaiUserMgr : paiUserMgr_typ := (0);
END_VAR
```

### Program Logical/paiComponents/paiUser/paiUser (ANSIC) - pai User Service (TK#8)

#### paiUser.c - Cyclic code
```c
#include <bur/plctypes.h>

#ifdef _DEFAULT_INCLUDES
	#include <AsDefault.h>
#endif

/*
###############################################################################
PAI_CONFIGURATION_SECTION
Code below allows configuration for:
User access
###############################################################################
*/
#warning "pai Configuration: User Access"

//=============================================================================
//User Login support
//=============================================================================
static void paiUserInitGroups()
{
	int ii;
	int groupIndex;

	gPaiUserConfig.loginTime_sec = 60.0 * 30.0;//30 minutes

	groupIndex = 0;
	brsstrcpy((UDINT)gPaiUserConfig.listGroups[groupIndex].Name, (UDINT)"NotLogged");
	gPaiUserConfig.listGroups[groupIndex].Level = 0;
	gPaiUserConfig.listGroups[groupIndex].Admin = 0;
	for(ii=0; ii<=paiUSER_RIGHTSMAXIDX;ii++){
		gPaiUserConfig.listGroups[groupIndex].AccessRights[ii] = mpUSER_ACCESS_UNDEFINED;
	}

	groupIndex = 1;
	brsstrcpy((UDINT)gPaiUserConfig.listGroups[groupIndex].Name, (UDINT)"Operator");
	gPaiUserConfig.listGroups[groupIndex].Level = 10;
	gPaiUserConfig.listGroups[groupIndex].Admin = 0;
	for(ii=0; ii<=paiUSER_RIGHTSMAXIDX;ii++){
		gPaiUserConfig.listGroups[groupIndex].AccessRights[ii] = mpUSER_ACCESS_FULL;
	}

	groupIndex = 2;
	brsstrcpy((UDINT)gPaiUserConfig.listGroups[groupIndex].Name, (UDINT)"Maintenance");
	gPaiUserConfig.listGroups[groupIndex].Level = 20;
	gPaiUserConfig.listGroups[groupIndex].Admin = 0;
	for(ii=0; ii<=paiUSER_RIGHTSMAXIDX;ii++){
		gPaiUserConfig.listGroups[groupIndex].AccessRights[ii] = mpUSER_ACCESS_FULL;
	}

	groupIndex = 3;
	brsstrcpy((UDINT)gPaiUserConfig.listGroups[groupIndex].Name, (UDINT)"Supervisor");
	gPaiUserConfig.listGroups[groupIndex].Level = 30;
	gPaiUserConfig.listGroups[groupIndex].Admin = 0;
	for(ii=0; ii<=paiUSER_RIGHTSMAXIDX;ii++){
		gPaiUserConfig.listGroups[groupIndex].AccessRights[ii] = mpUSER_ACCESS_FULL;
	}

	groupIndex = 4;
	brsstrcpy((UDINT)gPaiUserConfig.listGroups[groupIndex].Name, (UDINT)"Manufacturer");
	gPaiUserConfig.listGroups[groupIndex].Level = 100;
	gPaiUserConfig.listGroups[groupIndex].Admin = 1;
	for(ii=0; ii<=paiUSER_RIGHTSMAXIDX;ii++){
		gPaiUserConfig.listGroups[groupIndex].AccessRights[ii] = mpUSER_ACCESS_FULL;
	}

}

static void paiUserUpdatePWDUI()
{
	int ii;

	brsstrcpy((UDINT)gPaiUserMgr.userMgr.UIConnect.listUserNames[0]  ,(UDINT)"n.a.");
	brsstrcpy((UDINT)gPaiUserMgr.userMgr.UIConnect.listUserPasswords[0], (UDINT)"not used PIN");
	for(ii = 1; ii <=(paiUSER_USERSMAXIDX+1); ii++){
		brsstrcpy((UDINT)gPaiUserMgr.userMgr.UIConnect.listUserNames[ii]  ,(UDINT)gPaiUserConfig.listUsers[ii-1].UserName);
		brsitoa((UDINT)gPaiUserConfig.listUsers[ii-1].PIN, (UDINT)gPaiUserMgr.userMgr.UIConnect.listUserPasswords[ii] );
	}

}

static void paiUserInitUsers()
{
	int userIndex;

	userIndex = 0;
	brsstrcpy((UDINT)gPaiUserConfig.listUsers[userIndex].UserName, (UDINT)"Operator");
	brsstrcpy((UDINT)gPaiUserConfig.listUsers[userIndex].UserFullName, (UDINT)"Mach. Operator");
	gPaiUserConfig.listUsers[userIndex].PIN = 24025;
	gPaiUserConfig.listUsers[userIndex].GroupIndex = 1;

	userIndex = 1;
	brsstrcpy((UDINT)gPaiUserConfig.listUsers[userIndex].UserName, (UDINT)"Maintenance");
	brsstrcpy((UDINT)gPaiUserConfig.listUsers[userIndex].UserFullName, (UDINT)"Mach. Maintenance");
	//gPaiUserConfig.listUsers[userIndex].PIN = 9375144;
	gPaiUserConfig.listUsers[userIndex].PIN = 4858418;//changed on 9/21/2016, request from customer
	gPaiUserConfig.listUsers[userIndex].GroupIndex = 2;

	userIndex = 2;
	brsstrcpy((UDINT)gPaiUserConfig.listUsers[userIndex].UserName, (UDINT)"ABC Service");
	brsstrcpy((UDINT)gPaiUserConfig.listUsers[userIndex].UserFullName, (UDINT)"ABC Pckg.");
	gPaiUserConfig.listUsers[userIndex].PIN = 81134689;
	gPaiUserConfig.listUsers[userIndex].GroupIndex = 4;

//	userIndex = 3;
//	brsstrcpy(gPaiUserConfig.listUsers[userIndex].UserName, "user4");
//	brsstrcpy(gPaiUserConfig.listUsers[userIndex].UserFullName, "User Four");
//	gPaiUserConfig.listUsers[userIndex].PIN = 4444;
//	gPaiUserConfig.listUsers[userIndex].GroupIndex = 4;

	gPaiUserMgr.userMgr.UIConnect.userIndex = 0;
	gPaiUserMgr.userMgr.UIConnect.userIndexMax = userIndex;

	paiUserUpdatePWDUI();
}

static void	paiUserMgrInit()
{
	gPaiUserMgr.pUserConfig = &gPaiUserConfig;

	gPaiUserMgr.userMgr.UIConnect.pwdLevel = 0;
	gPaiUserMgr.userMgr.UIConnect.pwdLevelOld = 0;
	gPaiUserMgr.userMgr.UIConnect.visibleNotLogged = 0;//visible
	gPaiUserMgr.userMgr.UIConnect.visibleLogged = 1;//not visible
	gPaiUserMgr.userMgr.UIConnect.loggedIndex = 0;
	gPaiUserMgr.userMgr.UIConnect.isUserLogged = 0;

	brsmemcpy((UDINT)&gPaiUserMgr.currentGroup, (UDINT)&gPaiUserConfig.listGroups[0], sizeof(gPaiUserMgr.currentGroup));
	brsmemset((UDINT)&gPaiUserMgr.currentUser, 0, sizeof(gPaiUserMgr.currentUser));
	brsstrcpy((UDINT)gPaiUserMgr.currentUser.UserName  ,(UDINT)"n.a.");
	brsstrcpy((UDINT)gPaiUserMgr.currentUser.UserFullName, (UDINT)"n.a.");

}

static void paiUserMgrCyclic()
{

	//user login activity from the login screen
	if(gPaiUserMgr.userMgr.UIConnect.pwdLevel != gPaiUserMgr.userMgr.UIConnect.pwdLevelOld){
		if(gPaiUserMgr.userMgr.UIConnect.pwdLevel == (gPaiUserMgr.userMgr.UIConnect.userIndex + 1) ){
			//user login success!
			gPaiUserMgr.userMgr.UIConnect.isUserLogged = 1;

			gPaiUserMgr.userMgr.UIConnect.loggedIndex = gPaiUserMgr.userMgr.UIConnect.userIndex;
			if(gPaiUserMgr.userMgr.UIConnect.loggedIndex > paiUSER_USERSMAXIDX){
				gPaiUserMgr.userMgr.UIConnect.loggedIndex = paiUSER_USERSMAXIDX;
			}

			gPaiUserMgr.userMgr.UIConnect.visibleNotLogged = 1;//not visible
			gPaiUserMgr.userMgr.UIConnect.visibleLogged = 0;//visible visible

			//define current user
			brsmemcpy((UDINT)&gPaiUserMgr.currentUser, (UDINT)&gPaiUserConfig.listUsers[gPaiUserMgr.userMgr.UIConnect.loggedIndex], sizeof(gPaiUserMgr.currentUser));

			//define current group
			if(gPaiUserMgr.currentUser.GroupIndex > paiUSER_GROUPMAXIDX){
				gPaiUserMgr.currentUser.GroupIndex = paiUSER_GROUPMAXIDX;
			}
			brsmemcpy((UDINT)&gPaiUserMgr.currentGroup, (UDINT)&gPaiUserConfig.listGroups[gPaiUserMgr.currentUser.GroupIndex], sizeof(gPaiUserMgr.currentGroup));

			//start timeout timer
			bgTimerStart(&gPaiUserMgr.userMgr.loginTimer, 1000 * gPaiUserMgr.pUserConfig->loginTime_sec);
		}else{
			paiUserMgrInit();
		}
	}
	gPaiUserMgr.userMgr.UIConnect.pwdLevelOld = gPaiUserMgr.userMgr.UIConnect.pwdLevel;

	//login timer expired?
	if(gPaiUserMgr.userMgr.UIConnect.isUserLogged && bgTimerIsTimeOut(&gPaiUserMgr.userMgr.loginTimer) ){
		paiUserMgrInit();
	}

	//restart login timer button pressed?
	if(gPaiUserMgr.userMgr.UIConnect.btnRestartLoginTimer){
		gPaiUserMgr.userMgr.UIConnect.btnRestartLoginTimer = 0;
		bgTimerStart(&gPaiUserMgr.userMgr.loginTimer, 1000 * gPaiUserMgr.pUserConfig->loginTime_sec);
	}

	//login button pressed?
	if(gPaiUserMgr.userMgr.UIConnect.btnToggleLogin){
		gPaiUserMgr.userMgr.UIConnect.btnToggleLogin = 0;
		if(gPaiUserMgr.userMgr.UIConnect.isUserLogged){
			paiUserMgrInit();
		}else{
			//TODO: jump to login page
			gPaiHmiMain.runtime.pageChange = 70;//login page
		}
	}

	//operate login timer
	bgTimerCyclic(&gPaiUserMgr.userMgr.loginTimer);

	//calculate remaining login time [min:sec] from remaining timer time [ms]
	gPaiUserMgr.userMgr.UIConnect.remainingLoginTime_sec = 	( bgTimerTimeRemaining(&gPaiUserMgr.userMgr.loginTimer) / 1000 ) % 60;
	gPaiUserMgr.userMgr.UIConnect.remainingLoginTime_min = 	( bgTimerTimeRemaining(&gPaiUserMgr.userMgr.loginTimer) / 1000 ) / 60;
}

//=============================================================================

void _INIT paiUserInit(void)
{
	paiUserInitGroups();
	paiUserInitUsers();
	paiUserMgrInit();

}

void _CYCLIC paiUserCyclic(void)
{
	paiUserMgrCyclic();
}
//EOF
```

### paiBnRHW.typ
```iecst
(********************************************************************
 * COPYRIGHT --
 ********************************************************************
 * Package: paiComponents
 * File: paiBRHW.typ
 * Author: goran
 * Created: June 23, 2015
 ********************************************************************
 * Data types of package paiTelnet
 ********************************************************************)

TYPE
	paiBnRHWModuleInfo_typ : 	STRUCT
		ModuleOk : BOOL;
		SerialNumber : UDINT;
		ModuleID : UINT;
		HardwareVariant : UINT;
		FirmwareVersion : UINT;
	END_STRUCT;
END_TYPE
```

### Package Logical/Globals - application types and global vars

### Messages.typ - application alarms
```iecst
(********************************************************************

 * COPYRIGHT -- Piedmont Automation Inc.

 ********************************************************************

 * File: Alarms.typ

 * Author: goran

 * Created: Jun 1, 2015

 ********************************************************************

 * Data types for project : Alarms

 ********************************************************************)

TYPE
	applicationMessages_enums :
		(
		APP_MSG_READY := 0,
		APP_MSG_RUNAUTO,
		APP_MSG_RUNDRYCYCLE,
		APP_MSG_ZEROREQUIRED,
		APS_MSG_LOWONPALLETS,
		APP_MSG_ZERO_CASETURNER,
		APP_MSG_ZERO_ROWPUSHER,
		APP_MSG_ZERO_BLADESTOP,
		APP_MSG_ZERO_TABLE,
		APP_MSG_ZERO_ELEVATOR,
		APP_MSG_ZERO_PALLETELIFT,
		APP_MSG_ZERO_RETAINERBAR,
		APP_MSG_ZERO_SQUARING,
		APP_MSG_PALLETE_COMPLETE,
		APP_MSG_DISCHARGE_BLOCKED,
		APP_MSG_STOP_BLOCK_RT,
		APP_MSG_STOP_BLOCK_LF,
		APP_MSG_PALLETE_EXITING,
		APP_MSG_ZERO_MSG18,
		APP_MSG_ZERO_MSG19,
		APP_MSG_LAST := 50
		);
END_TYPE

(*########################################################################*)
(*Application object - Message Object*)
(*########################################################################*)

TYPE
	applicationMessages_typ : 	STRUCT
		oIsMsgActive : BOOL; (*1-if alarm present*)
		msgActive : ARRAY[0..APP_MSG_LAST]OF BOOL; (*Alarms matrix. (see Visual Components Alarm System)*)
	END_STRUCT;
END_TYPE
```

### Messages.var
```iecst
(*********************************************************************************
 * Copyright: Piedmont Automation Inc
 * Author:    Goran
 * Created:   Jun 26, 2015/11:38 AM
 *********************************************************************************
 * Declaration of global variables
 *********************************************************************************)
VAR
	gMsgScroll : paiHmiMsgScrolling_typ := (0); (*Scrolling Alarm Msg Support*)
	gMessages : applicationMessages_typ := (0);
END_VAR
```

### MachineVFD.var
```iecst
(*********************************************************************************
 * Copyright: Piedmont Automation Inc
 * Author:    Goran
 * Created:   Jun 26, 2015/11:38 AM
 *********************************************************************************
 * Declaration of global variables
 *********************************************************************************)
VAR
	gMachineVFD : ARRAY[0..APP_VFD_IDXLAST] OF paiVFD_typ;
END_VAR
```

### ConfigApp.typ - Global types - machine configuration - application level - CHANGE AS NEEDED
```iecst
(********************************************************************
 * COPYRIGHT --
 ********************************************************************
 * Package: ConfigAndRecipes
 * File: appConfig.typ
 * Author: goran_2
 * Created: August 06, 2011

DEFINE APPLICATION SPECIFIC CONFIG STRUCTURES AS NEEDED

(*Insert your comment here.*)

TYPE
	appCfgEnums_typ :
		(
		New_Member
		);
	appCfgTimers_typ : 	STRUCT
		dlyTableLayerRdyToElevMove : REAL; (*delay from table layer ready before elevator moves*)
		dlyTableAtPalleteToRetBar : REAL; (*delay from table at pallete before retainter bar lowered*)
		onDlyPRRetBarDown : REAL; (*on delay for Retainer Bar Down prox switch*)
		onTmCaseTurner : REAL; (*case turner dwell time*)
		onDlyEEPallete : REAL; (*on delay for pallete/box detection PE EE2*)
		offDlyEEPallete : REAL; (*off delay for pallete/box detection PE EE2*)
		onDlyPRRetBarDown2 : REAL; (*on delay for Retainer Bar Down prox switch*)
		dlyLastCaseToRowCVStop : REAL; (*delay from Row forming complete to row push. Needed to allow box to travel.*)
		dlyRowDoneToRowPush : REAL; (*delay from Row forming complete to row push. Needed to allow box to travel.*)
		infeedCVIdleTime : REAL; (*max allowed time to run infeed cv-s before stopping them*)
		JamAlarmTmAtInfeedEE2 : REAL;
		JamAlarmTmAtRowToLongEE8 : REAL;
		JamAlarmTmRowForming : REAL;
		onDlyPalleteDischargeEE16 : REAL; (*on delay for pallete discharge sensor; longer time adjustst position of the pallete pass the sensor*)
		palletExitAlarmTm : REAL; (*pallet exit alarm time*)
		EE2OnDebounce : REAL;
		EE2OfDebounce : REAL;
		EE4OnDebounce : REAL;
		EE4OfDebounce : REAL;
		EE8OnDebounce : REAL;
		EE8OfDebounce : REAL;
		EE16OfDebounce : REAL;
		dlyPusherAtElevatorToRetract : REAL; (*dealy from pusher at extended position (et elevator) to trigger retracted motion *)
		onDlyFrontSquaring : REAL;
		onDlyTableToGrouping : REAL; (*on delay after layer is dropped onto the paller before table is moved back to grouping*)
		onDlyRetBarDown : REAL; (*On delay from the moment table starts moving to the pallet before retainer bar is lowered*)
		bladeStopOnDly1 : REAL; (*Blade stop turn on delay time; to accomoated for case traveling on the row forming belt*)
		bladeStopOnDly2 : REAL; (*Blade stop turn on delay time; to accomoated for case traveling on the row forming belt*)
		bladeStopOnDly3 : REAL; (*Blade stop turn on delay time; to accomoated for case traveling on the row forming belt*)
		bladeStopOnDly4 : REAL; (*Blade stop turn on delay time; to accomoated for case traveling on the row forming belt*)
		bladeStopOnDly5 : REAL; (*Blade stop turn on delay time; to accomoated for case traveling on the row forming belt*)
		bladeStopOnDly6 : REAL; (*Blade stop turn on delay time; to accomoated for case traveling on the row forming belt*)
	END_STRUCT;
	appCfgOptions_typ : 	STRUCT
		optTearSheetEquiped : UDINT; (*1-Tear sheet insert mechanism is present*)
		optOption1Equiped : UDINT; (*1-Tear sheet insert mechanism is present*)
		palletDispenserOption : UDINT; (*0-pallet dispenser is NOT present/NOTequipped; 1-pallet dispenser option IS present/equipped*)
		frontSquaringOption : UDINT; (*0-front squaring option is NOT present/NOTequipped; 1-front squaring option is present*)
		dryCycleCaseCount : UDINT;
		dryCycleRowCount : UDINT;
		dryCycleLayerCount : UDINT;
		tmDryCycleElevatorUp : REAL; (*time to dry cycle operation to simulate layers*)
		tmDryCycleCaseTime : REAL; (*single case loading time in dry cycle simulation*)
		dryCycleLayerDonePause : UDINT;
		tmDryCycleLayerZeroOffset : REAL; (*single case loading time in dry cycle simulation*)
	END_STRUCT;
	appCfgSystem_typ : 	STRUCT
		bladeStopCount : UDINT; (*number of blade stops (0...6)*)
		simulationMode : UDINT; (*1-yes*)
		bladeStopOnDly : ARRAY[0..APP_CFG_BLADESTOP_MAXIDX]OF REAL; (*Blade stop turn on delay time; to accomoated for case traveling on the row forming belt*)
		bladeStopDistance : ARRAY[0..APP_CFG_BLADESTOP_MAXIDX]OF REAL; (*Blade stop distance[inch]*)
		boxInfeedSide : UDINT; (*0-infeed from left to right 1-infeed from right to left; point of refernece if front of the machine infeed looking towards the table*)
	END_STRUCT;
	cfgMachineVFDs_typ : 	STRUCT
		velocitySlow_rpm : DINT; (*slow velocity (if needed)*)
		velocity_rpm : DINT; (*normal velocity*)
		acc : DINT; (*accelaration [x0.1sec]*)
		dec : DINT; (*decelaration [x0.1sec]*)
	END_STRUCT;
END_TYPE

(*######################################################*)

TYPE
	configApp_typ : 	STRUCT  (*Machine configuration includes settings for timers and settings for servo drives.*)
		system : appCfgSystem_typ;
		options : appCfgOptions_typ;
		magicNumber : UDINT;
	END_STRUCT;
END_TYPE
```

### Defaults_gConfigApp.c
```c
/********************************************************************
 * COPYRIGHT -- piedmont
 ********************************************************************
 * Program: Defaults_gConfigApp
 * File: Defaults_gConfigApp.c
 * Author: admin
 * Created: Jan 20, 2015
 ********************************************************************
 * Implementation of program Defaults_gConfigApp
 ********************************************************************/

#include <bur/plctypes.h>

#ifdef _DEFAULT_INCLUDES
 #include <AsDefault.h>
#endif

/*
###############################################################################
PAI_CONFIGURATION_SECTION
Code below allows configuration of the PV serialization / deserialization
manager.
###############################################################################
*/
#warning "app Configuration: PV Defaults for gConfigApp"

void gConfigAppDefaults()
{
int ii;

	gConfigApp.options.dryCycleCaseCount = 5;
	gConfigApp.options.dryCycleLayerCount = 3;
	gConfigApp.options.dryCycleLayerDonePause = 0;
	gConfigApp.options.palletDispenserOption = 1;
	gConfigApp.options.dryCycleRowCount = 4;
	gConfigApp.options.tmDryCycleCaseTime = 2.0;
	gConfigApp.options.tmDryCycleElevatorUp = 3.0;
	gConfigApp.options.tmDryCycleLayerZeroOffset = 2.0;

	gConfigApp.system.simulationMode = 0;
	gConfigApp.system.boxInfeedSide = 0;
	gConfigApp.system.bladeStopCount = 1;
	gConfigApp.system.bladeStopDistance[0] = 6.0;
	gConfigApp.system.bladeStopDistance[1] = 8.0;
	gConfigApp.system.bladeStopDistance[2] = 10.0;
	gConfigApp.system.bladeStopDistance[3] = 12.0;
	gConfigApp.system.bladeStopDistance[4] = 14.0;
	gConfigApp.system.bladeStopDistance[5] = 16.0;

}

void gPalletCfgDefaults()
{
	int ii;

	gPallete.palCfg.palSettings.timers.dlyTableAtPalleteToRetBar = 1.0;
	gPallete.palCfg.palSettings.timers.dlyTableLayerRdyToElevMove = 1.0;
	gPallete.palCfg.palSettings.timers.offDlyEEPallete = 1.0;
	gPallete.palCfg.palSettings.timers.onDlyPRRetBarDown = 1.0;
	gPallete.palCfg.palSettings.timers.onDlyPRRetBarDown2 = 1.0;
	gPallete.palCfg.palSettings.timers.onTmCaseTurner = 1.0;
	gPallete.palCfg.palSettings.timers.dlyRowDoneToRowPush = 1.0;
	gPallete.palCfg.palSettings.timers.dlyTableAtPalleteToRetBar = 1.0;
	gPallete.palCfg.palSettings.timers.JamAlarmTmAtInfeedEE2 = 4.0;
	gPallete.palCfg.palSettings.timers.JamAlarmTmRowForming = 4.0;
	gPallete.palCfg.palSettings.timers.JamAlarmTmAtRowToLongEE8 = 4.0;
	gPallete.palCfg.palSettings.timers.palletExitAlarmTm = 10.0;
	gPallete.palCfg.palSettings.timers.infeedCVIdleTime = 15.0;
	gPallete.palCfg.palSettings.timers.onDlyPalleteDischargeEE16 = 1.0;
	gPallete.palCfg.palSettings.timers.onDlyTableToGrouping = 0.0;
	gPallete.palCfg.palSettings.timers.EE2OfDebounce = 0.0;
	gPallete.palCfg.palSettings.timers.EE2OnDebounce = 0.0;
	gPallete.palCfg.palSettings.timers.EE4OfDebounce = 0.0;
	gPallete.palCfg.palSettings.timers.EE4OnDebounce = 0.0;
	gPallete.palCfg.palSettings.timers.EE8OfDebounce = 0.0;
	gPallete.palCfg.palSettings.timers.EE8OnDebounce = 0.0;
	gPallete.palCfg.palSettings.timers.EE16OfDebounce = 0.0;
	gPallete.palCfg.palSettings.timers.onDlyFrontSquaring = 0.0;
	gPallete.palCfg.palSettings.timers.bladeStopOnDly1 = 3.0;
	gPallete.palCfg.palSettings.timers.bladeStopOnDly2 = 3.0;
	gPallete.palCfg.palSettings.timers.bladeStopOnDly3 = 3.0;
	gPallete.palCfg.palSettings.timers.bladeStopOnDly4 = 2.0;
	gPallete.palCfg.palSettings.timers.bladeStopOnDly5 = 2.0;
	gPallete.palCfg.palSettings.timers.bladeStopOnDly6 = 2.0;

	for(ii=0; ii<=APP_VFD_IDXLAST; ii++){
		gPallete.palCfg.palSettings.vfd[ii].velocitySlow_rpm = 0.0;
		gPallete.palCfg.palSettings.vfd[ii].velocity_rpm = 0.0;
	}

	gPallete.palCfg.palSettings.vfd[1].velocitySlow_rpm = 300.0;
	gPallete.palCfg.palSettings.vfd[1].velocity_rpm = 600.0;
	gPallete.palCfg.palSettings.vfd[2].velocitySlow_rpm = 300.0;
	gPallete.palCfg.palSettings.vfd[2].velocity_rpm = 600.0;
	gPallete.palCfg.palSettings.vfd[4].velocitySlow_rpm = 300.0;
	gPallete.palCfg.palSettings.vfd[4].velocity_rpm = 600.0;
	gPallete.palCfg.palSettings.vfd[5].velocitySlow_rpm = 300.0;
	gPallete.palCfg.palSettings.vfd[5].velocity_rpm = 600.0;
	gPallete.palCfg.palSettings.vfd[6].velocitySlow_rpm = 300.0;
	gPallete.palCfg.palSettings.vfd[6].velocity_rpm = 600.0;
	gPallete.palCfg.palSettings.vfd[11].velocitySlow_rpm = 300.0;
	gPallete.palCfg.palSettings.vfd[11].velocity_rpm = 600.0;
	gPallete.palCfg.palSettings.vfd[12].velocitySlow_rpm = 300.0;
	gPallete.palCfg.palSettings.vfd[12].velocity_rpm = 600.0;

	for(ii=0; ii <= APP_VFD_IDXLAST; ii++){
		gPallete.palCfg.palSettings.vfd[ii].acc = 1;
		gPallete.palCfg.palSettings.vfd[ii].dec = 1;
	}

}
//EOF
```

### Package Logical/MachineControl - application tasks and logic

### MachineControl.typ - Global data types
```iecst
(*********************************************************************************
 * Copyright: Microsoft
 * Author:    Obed
 * Created:   May 26, 2015/11:38 AM
 *********************************************************************************
 * Declaration of AppControl global data types for ABC Palletizer
 *********************************************************************************)
(*********************************************************************************
	Application Structures
*********************************************************************************)

TYPE
	macCtrlEnums_typ :
		(
		APP_REC_MAXCASE := 12, (*Max number of cases per row*)
		APP_REC_MAXROW := 12, (*Max number of rows per layer*)
		APP_REC_MAXLAYER := 12 (*Max number of layers per palette*)
		);
END_TYPE

(*********************************************************************************
macCtrl_typ Contains all machine Control Structures. Using "mac" as abbreviation for Machine, "Ctrl" as for Control
*********************************************************************************)

TYPE
	macCtrl_typ : 	STRUCT
		main : macCtrlMain_typ; (*Machine Main*)
		infeedcv : macCtrlInfeedCV_typ; (*Timing Infeed Conveyor*)
		rowforming : macCtrlRowForming_typ; (*Row Forming Conveyor*)
		caseturner : macCtrlCaseTurner_typ; (*Case Turner*)
		retainerbar : macCtrlRetainerBar_typ;
		transfertable : macCtrlTransferTable_typ; (*Roller Transfer Table*)
		squaring : macCtrlSquaringPlates_typ; (*Main Frame Side Squaring Plates*)
		elevator : macCtrlElevator_typ; (*Main Frame Elevator*)
		palletDispenser : macCtrlPalleteDispenser_typ; (*Pallet Dispenser*)
		palletDischarge : macCtrlPalleteDischarge_typ; (*Pallet Dispenser*)
	END_STRUCT;
END_TYPE

(*********************************************************************************
macCtrlMain_typ Machine Main
*********************************************************************************)

TYPE
	macCtrlMain_typ : 	STRUCT
		modeMaintenance : BOOL; (*Mode: service/maintance. Minor or Major Fault active. Start (Auto) not possible.*)
		modeManual : BOOL; (*Mode: manual; No faults. Not in auto mode. Buttons to start auto mode IS available.*)
		modeAuto : BOOL; (*Mode: auto is active. See below for available auto modes.*)
		modeAutoProduction : BOOL; (*Mode: autoProduction; Auto. Production, Normal operation. Button to stop is available.*)
		modeAutoDryCycle : BOOL; (*Mode: autoDryCycle; Auto. DryCycleMode, Testing option. Button to stop is available.*)
		modeAutoDemo : BOOL; (*Mode: autoDemo; Auto. Demp/Show mode, Used for Show. Button to stop is available.*)
		modeAutoStarting : BOOL; (*Mode: autoStarting; Auto. Transitioning from Manual to Auto. (i.e. Start Button Pressed).*)
		modeAutoStopping : BOOL; (*Mode: autoStopping; Auto. Transitioning from Auto to Manual. (i.e. Stop Button Pressed).*)
		buttonEnabledStart : BOOL; (*Start Button control.*)
		buttonEnabledMaint : BOOL; (*Start Button control.*)
		noMajorFault : BOOL; (*No major fault on the machine.*)
		noMinorFault : BOOL; (*No minor fault on the machine.*)
		noFaults : BOOL; (*No minor or major fault on the machine.*)
		guardDoorsOk : BOOL; (*Guard door safety indicator.*)
		EStopOk : BOOL; (*EStop safety indicator.*)
		SafetyOk : BOOL; (*Safety Circuit OK*)
		VFDsNoFaults : BOOL; (*VFDs fault indication*)
		isAtZero : BOOL; (*machine is at zero position*)
		zeroIsNeeded : BOOL; (*machine is at zero position*)
		btnZero : BOOL; (*0-not pressed; 1-presed*)
		btnStart : BOOL; (*0-not pressed; 1-presed*)
		btnStop : BOOL; (*0-not pressed; 1-presed*)
		btnFaultAck : BOOL; (*1-ack fault / alarms*)
		btnClearCaseCounts : BOOL; (*1-ack fault / alarms*)
		btnZeroVisibility : INT; (*0-visible; 1-not visible*)
		hmiShowMsgZeroingNeeded : BOOL;
		btnNotInAutoModeVisibility : INT; (*0-visible; 1-not visible*)
		btnStartVisibility : INT; (*0-visible; 1-not visible*)
		btnLoadMachineCfg : BOOL;
		alwaysOnBit : BOOL; (*Always on bit*)
		testBit1 : BOOL; (*Test bit 1: TESTING ONLY! REMOVE FROM A FINAL PROGRAM!*)
		testBit2 : BOOL; (*Test bit 2: TESTING ONLY! REMOVE FROM A FINAL PROGRAM!*)
		testBit3 : BOOL; (*Test bit 3: TESTING ONLY! REMOVE FROM A FINAL PROGRAM!*)
		dummyCoil : BOOL; (*Dummy coil*)
		blink : BOOL; (*Light on/off blink signal*)
		gCamApp_btnPreview : BOOL;
		optionEStops : ARRAY[0..5]OF BOOL; (*Configuration Option for EStops Circuits*)
		optionDoorSw : ARRAY[0..5]OF BOOL; (*Configuration Options of Door Safety Switches*)
		visibleCaseInfeedOnLeft : UDINT; (*Visibility control for HMI when Case infeed on the left*)
		visibleCaseInfeedOnRight : UDINT; (*Visibility control for HMI when Case infeed on the right*)
		isDropLayerToPalletAllowed : BOOL;
		dropLayerToPalletBlock : BOOL;
		elevatorStopBlockActive : BOOL; (*Elevator stops blocks are active. This is part of the safety logic. *)
		tmrMCROnDelay : TON; (*Timer for MCR on delay*)
		tmrAirOnDelay : TON; (*Timer for air on delay*)
		tmrBlinkOn : TON; (*Timer for blink signal*)
		tmrBlinkOff : TOF; (*Timer for blink signal*)
	END_STRUCT;
END_TYPE

(*********************************************************************************
macCtrlMode_typ Machine Control Modes of Operation
*********************************************************************************)

TYPE
	macCtrlMode_typ : 	STRUCT
		Maintenance : BOOL; (*Minor or Major Fault active*)
		Manual : BOOL; (*Not in auto mode. Buttons to start auto mode are available.*)
		AutoProduction : BOOL; (*Auto. Production, Normal operation. Button to stop is available.*)
		AutoDryCycle : BOOL; (*Auto. DryCycleMode, Testing option. Button to stop is available.*)
		AutoDemo : BOOL; (*Auto. Demp/Show mode, Used for Show. Button to stop is available.*)
		AutoStarting : BOOL;
		AutoStopping : BOOL;
	END_STRUCT;
END_TYPE

(*********************************************************************************
macCtrlStats_typ Machine Statistics data (case counts, etc)
*********************************************************************************)

TYPE
	macCtrlStats_typ : 	STRUCT
		btnResetCounts : BOOL;
		btnResetCountsTotal : BOOL;
		casesPerMin : UDINT;
		caseCounter : UDINT;
		caseCounterTotal : UDINT;
		palletCounter : UDINT;
		palletCounterTotal : UDINT;
		palletTimeMin : REAL;
		palletTimeMax : REAL;
		palletTimeLast : REAL;
		runningTmr1 : TON;
		runningTmr1min : TON;
		runningTmr1sec : TON;
		palletTmr : TON;
		runTmrHours : UDINT;
		runTmrMins : UDINT;
		runTmrSec : UDINT;
		mCasesPerMinCounter : UDINT;
	END_STRUCT;
END_TYPE

(*********************************************************************************
macCtrlTimingInfeedConveyor_typ #TIMING INFEED CONVEYOR
*********************************************************************************)

TYPE
	macCtrlInfeedCV_typ : 	STRUCT
		hmiBtnOnOff : BOOL;
		infeedCvOn : BOOL;
		caseInSensorNegEdge : BOOL;
		caseInSensorPosEdge : BOOL;
		caseInSensor : BOOL;
		caseOutSensorNegEdge : BOOL;
		caseOutSensorPosEdge : BOOL;
		caseOutSensor : BOOL;
		caseAtOneCaseOnlySection : BOOL;
		nextCaseToCloseMonitorEnabled : BOOL;
		caseInfeedDone : BOOL;
		tmrJamAtCaseInSensorEE2 : TON;
		tmrJamAtCaseStageSensorEE4 : TON;
		tmrJamAtCaseOutSensorEE8 : TON;
		tmrJamRowForming : TON;
		tmrInfeedCVIdle : TON;
		tmrInfeedStopDly : TON;
		rowFormingCVRunPosEdge : BOOL;
		rowFormingCVRunNegEdge : BOOL;
		ssmInfeedCV : bgSSM_typ;
		sleepState : BOOL;
		stopRequest : BOOL;
	END_STRUCT;
END_TYPE

(*********************************************************************************
macCtrlRowFormingConveyor_typ #ROW FORMING CONVEYOR
*********************************************************************************)

TYPE
	macCtrlRowForming_typ : 	STRUCT
		isRowPusherAtHome : BOOL;
		isRowPusherAtElevator : BOOL;
		hmiBtnPusherFwdJog : BOOL;
		hmiBtnPusherRevJog : BOOL;
		hmiBtnPusherFwd : BOOL;
		hmiBtnPusherRev : BOOL;
		hmiBtnOnOffStageCV : BOOL;
		hmiBtnOnOffCV : BOOL;
		hmiBtnStopBladeUpDown1 : BOOL;
		hmiBtnStopBladeUpDown2 : BOOL;
		hmiBtnStopBladeUpDown3 : BOOL;
		hmiBtnStopBladeUpDown4 : BOOL;
		hmiBtnStopBladeUpDown5 : BOOL;
		hmiBtnStopBladeUpDown6 : BOOL;
		hmiBtnStopBladeUpDownQuick1 : BOOL;
		hmiBtnStopBladeUpDownQuick2 : BOOL;
		hmiBtnStopBladeUpDownQuick3 : BOOL;
		hmiBtnStopBladeUpDownQuick4 : BOOL;
		hmiBtnStopBladeUpDownQuick5 : BOOL;
		hmiBtnStopBladeUpDownQuick6 : BOOL;
		New_Member : USINT;
		isStopBladeUsed1 : BOOL;
		isStopBladeUsed2 : BOOL;
		isStopBladeUsed3 : BOOL;
		isStopBladeUsed4 : BOOL;
		isStopBladeUsed5 : BOOL;
		isStopBladeUsed6 : BOOL;
		allBladesDown : BOOL;
		lastCaseToStopCVDly : TON;
		rowPusherOnDly : TON;
		bladeStopOnDly : ARRAY[0..5]OF TON;
	END_STRUCT;
END_TYPE

(*********************************************************************************
macCtrlCaseTurner_typ #CASE TURNER
*********************************************************************************)

TYPE
	macCtrlCaseTurner_typ : 	STRUCT
		hmiBtnCaseTurnerUpDown : BOOL;
		hmiAutoCaseTurn : BOOL; (*0-no case turn; 1-case turn (raise turner)*)
		tmrCaseTurnerActive : TON;
	END_STRUCT;
END_TYPE

(*********************************************************************************
macCtrlRollerTransferTable_typ #ROLLER TRANSFER TABLE
*********************************************************************************)

TYPE
	macCtrlTransferTable_typ : 	STRUCT
		isTableAtGrouping : BOOL;
		isTableAtPallete : BOOL;
		hmiBtnTableFwdJog : BOOL;
		hmiBtnTableRevJog : BOOL;
		hmiBtnTableFwd : BOOL;
		hmiBtnTableRev : BOOL;
		hmiBtnOnOffCV : BOOL;
	END_STRUCT;
	macCtrlRetainerBar_typ : 	STRUCT
		revTimer : TON;
		fwdTimer : TON;
		barDwOffDlyTmr : TON;
		barDwDlyTmXms : UDINT;
		barIsUp : BOOL;
		barIsDown : BOOL;
		hmiBtnRetainterBarFwdJog : BOOL;
		hmiBtnRetainterBarRevJog : BOOL;
		hmiBtnRetainterBarFwd : BOOL;
		hmiBtnRetainterBarRev : BOOL;
	END_STRUCT;
END_TYPE

(*********************************************************************************
macCtrlElevator_typ #MAIN FRAME ELEVATOR
*********************************************************************************)

TYPE
	macCtrlElevator_typ : 	STRUCT
		elevatorIsAtTop : BOOL; (*Elevator at home position*)
		elevatorIsAboveHomeUnknown : BOOL; (*Elevator above home*)
		elevatorIsAboveNearHome : BOOL; (*Elevator above home*)
		elevatorIsAboveHome : BOOL; (*Elevator above home*)
		elevatorIsAtHome : BOOL; (*Elevator at home position*)
		elevatorIsBelowHome : BOOL; (*Elevator is below home position*)
		elevatorIsBelowNearHome : BOOL; (*Elevator is below home position*)
		elevatorIsBelowHomeUnknown : BOOL; (*Elevator is below home position, both switches out*)
		elevatorIsAtBottom : BOOL; (*Elevator at home position*)
		elevatorIsUknownPosition : BOOL; (*Elevator is below home position*)
		elevatorIsMovingUp : BOOL; (*Elevator is below home position*)
		elevatorIsMovingDw : BOOL; (*Elevator is below home position*)
		elevatorIsAtPalleteBelowHome : BOOL; (*Elevator is below home position*)
		elevatorIsAtPalleteAboveHome : BOOL; (*Elevator is below home position*)
		hmiBtnElevatorToHome : BOOL; (*Send elevator to home (which is grouping/loading position)*)
		hmiBtnElevatorToGrouping : BOOL; (*Send elevator to grouping/loading position*)
		hmiBtnElevatorToAbovePallete : BOOL; (*Send elevator to above the pallete for pallete exiting when front squaring option is present*)
		hmiBtnElevatorToPallete : BOOL; (*Send elevator to pallete top/unloading position*)
		hmiBtnElevatorToTop : BOOL; (*Send elevator to the top position*)
		hmiBtnElevatorFwdJog : BOOL; (*Jog Fwd (UP)*)
		hmiBtnElevatorRevJog : BOOL; (*Jog Rev (DW)*)
		hmiBtnElevatorFwd : BOOL; (*Move Fwd (UP to the top)*)
		hmiBtnElevatorRev : BOOL; (*Move Rev (DW to the bottom)*)
		tmrPalletePEOff : TOF;
		tmrPalletePEOn : TON;
	END_STRUCT;
END_TYPE

(*********************************************************************************
macCtrlSideSquaringPlates_typ #SIDE SQUARING PLATES
*********************************************************************************)

TYPE
	macCtrlSquaringPlates_typ : 	STRUCT
		frontSquaringEquipped : BOOL;
		hmiBtnFrontPlateExtRet : BOOL;
		hmiBtnSidePlatesExtRet : BOOL;
		tmrFrontSquaringOnDly : TON;
	END_STRUCT;
END_TYPE

(*********************************************************************************
macCtrlDispenser_typ #PALLET DISPENSER
*********************************************************************************)

TYPE
	macCtrlPalleteDispenserEnums_typ :
		(
		PLT_DISPENSE_ZERO := 0,
		PLT_DISPENSE_INIT,
		PLT_DISPENSE_IDLE,
		PLT_DISPENSE_TOBOTTOM,
		PLT_DISPENSE_WTCLAWSOPN,
		PLT_DISPENSE_TOMID,
		PLT_DISPENSE_WTCLAWSCLS,
		PLT_DISPENSE_DN
		);
	macCtrlPalleteDispenser_typ : 	STRUCT
		palletDispenserEquippedVis : USINT; (*0-visible when  equipped; 1-not visible when not equipped*)
		palletDispenserEquipped : BOOL; (*0-not equipped; 1-equipped*)
		hmiBtnPalletClawsOpenClose : BOOL;
		hmiBtnPalletInCVFwdJog : BOOL;
		hmiBtnPalletInCVRevJog : BOOL;
		hmiBtnPalletInCVFwd : BOOL;
		hmiBtnPalletInCVRev : BOOL;
		hmiBtnClawsLiftUpJog : BOOL;
		hmiBtnClawsLiftDwJog : BOOL;
		atTop : BOOL;
		atMidHi : BOOL;
		atMidLo : BOOL;
		atBottom : BOOL;
		flagClawsLiftToMidHi : BOOL;
		flagClawsLiftToMidLo : BOOL;
		flagMoveUp : BOOL;
		hmiBtnClawsLiftToTop : BOOL;
		hmiBtnClawsLiftToMidHi : BOOL;
		hmiBtnClawsLiftToMidLo : BOOL;
		hmiBtnClawsLiftToBottom : BOOL;
		dispenseState : macCtrlPalleteDispenserEnums_typ;
		dispenseReq : BOOL;
		dispenseIP : BOOL;
		dispenseDN : BOOL;
		clawsOpenTmr : TON;
	END_STRUCT;
	macCtrlPalleteDischarge_typ : 	STRUCT
		hmiBtnPalletDischargeCVFwdJog : BOOL;
		hmiBtnPalletDischargeCVRevJog : BOOL;
		hmiBtnPalletDischargeCVFwd : BOOL;
		hmiBtnPalletDischargeCVRev : BOOL;
		hmiBtnPalletManualExit : BOOL;
		palletManualExitRequest : BOOL;
		palletManualFinishRequest : BOOL;
		muteLightCurtainDuringDischarge : BOOL;
		dischargePESensor : BOOL;
		dischargeState : UDINT;
		dischargeReq : BOOL;
		isDischargeAllowed : BOOL;
		dischargeIP : BOOL;
		dischargeDN : BOOL;
		dischargeRecoveryIP : BOOL;
		dischargeRecoveryVisible2 : BOOL;
		dischargeRecoveryVisible : UINT;
		dischargePESensorTmrOf : TOF;
		dischargeMuteRecoveryTmr : TON;
		dischargeMuteTmr : TOF;
		dischargeTmr : TON;
		palleteExitTmoutTmr : TON;
	END_STRUCT;
END_TYPE

(*********************************************************************************
appControlLogic_typ
*********************************************************************************)

TYPE
	appControlLogic_typDELETE : 	STRUCT  (*Application Control*)
		cmd : appControlCmd_typ; (*Commands*)
		status : appMachineStatus_typ; (*Machine Status*)
		seekStartPosition : BOOL; (*Seek Start Position*)
		seekStartInAuto : BOOL; (*Seek Start In Auto*)
		seekStartInHand : BOOL; (*Seek Start In Hand*)
		autoCycleComplete : BOOL; (*Auto Cycle Complete*)
		handExitFullPallet : BOOL; (*Hand Exit Full Pallet*)
		handMode : BOOL; (*Hand Mode*)
		palletRunout : BOOL; (*Pallet Runout*)
		safetyCircuitEnergized : BOOL; (*Safety Circuit Energized*)
		guardDoorsOK : BOOL; (*Guard Doors OK*)
		guardDoor1Message : BOOL; (*Guard Door 1 Message*)
		guardDoor2Message : BOOL; (*Guard Door 2 Message*)
		guardDoor3Message : BOOL; (*Guard Door 3 Message*)
		guardDoor4Message : BOOL; (*Guard Door 4 Message*)
		dispenserGuardEyeMessage : BOOL; (*Dispenser Guard Eye Message*)
		machineHasPalletDispensor : BOOL; (*Machine Has Palllet Dispensor ???*)
		dischargeGuardEyeMessage : BOOL; (*Discharge Guard Eye Message*)
		inserterGuardEyeMessage : BOOL; (*Inserter Guard Eye Message*)
		Check_Drive1 : BOOL; (*Check Drive 1*)
		Check_Drive4 : BOOL; (*Check Drive 4*)
		Drive4_OverCurrent : BOOL; (*Drive 4 OverCurrent*)
		VFD_On_Row_Pusher : BOOL; (*VFD On Row Pusher*)
		rollerSleep : BOOL; (*Roller Sleep Reset ????*)
		machineHasServoOrTurnTable : BOOL; (*Machine Has Servo Or Turn Table #TURNER*)
		dryCycleMode : BOOL; (*Dry Cycle Mode*)
		runOut : BOOL; (*RunOut*)
		CheckDrive4TON : TON; (*Check Drive 4 TON*)
		DelayForDriveDischargeTON : TON; (*Delay For Drive Discharge TON*)
		DelayAirOnTON : TON; (*Delay For Air On TON*)
		CheckDrive1TON : TON; (*Check Drive 1TON*)
		MSROnDelayedTOF : TOF; (*MSR ON Delayed TOF*)
		CaseCountEyeOFFDelayTOF : TOF; (*Case Count Eye OFF Delay*)
		AutoCycleDelayOFF : BOOL; (*AutoCycleDelayOFF*)
		AutoCycleDelayOFFTOF : TOF; (*AutoCycleDelayOFF TOF*)
		RollerSleepTON : TON; (*Roller Sleep TON*)
		noDrive1Confirm : BOOL; (*No Drive 1 Confirm*)
		MSROnDelayed : BOOL; (*MSR On Delayed*)
		DelayForDriveDischarge : BOOL; (*Delay For Drive Discharge*)
		NoMinorFault : BOOL; (*No Minor Fault*)
		NoMajorFault : BOOL; (*No Major Fault*)
		NotOkOneShot : BOOL; (*Not Ok One Shot*)
		DelayForAirOn : BOOL; (*Delay For Air On*)
		noProductComming : BOOL; (*No Product Comming*)
		MotorOverloads : BOOL; (*Motor Overloads ???*)
		MachineHasCategory3Safety : BOOL; (*Machine has category 3 safety*)
		MachineHasAuxsVFDs : BOOL; (*Machine has Auxs VFDs ???*)
		MachineHasServoTurner : BOOL; (*Machine has Servo Turner SERVO_OPTION*)
		MachineHasBottomSheetInserter : BOOL; (*Machine has Bottom Sheet Inserter ???*)
		MachineHasOverHeadPusher : BOOL; (*Machine has Overhead Pusher ???*)
		MachineHasOverHeadInserter : BOOL; (*Machine has Overhead Inserter ???*)
		CountsDontMatch : BOOL; (*Counts Dont Match*)
		StartPosition : BOOL; (*Start Position*)
		ZeroMachine : BOOL; (*Zero Machine*)
		ResetLayer : BOOL; (*Reset Layer*)
		Pallet_Disch_BypassSelectorSW : BOOL; (*Pallet Discharge Bypass Selector Switch SS5 ???*)
		DownCount : BOOL; (*Down Count*)
		PushedEndOfRun : BOOL; (*Pushed End of Run*)
		RowPusherLeavingHome : BOOL; (*Row Pusher Leaving Home*)
		RowCountImpulse : BOOL; (*RowCountImpulse*)
		CaseCountEyeOFFDelay : BOOL; (*Case Count Eye OFF Delay*)
		CaseCountImpulse : BOOL; (*Case Count Impulse*)
		DontRunThisOne : BOOL; (*Don't Run This One*)
		SingleScan : BOOL; (*Single Scan*)
		ResetCaseCount : BOOL; (*Reset Case Counts*)
		BackOfLastBag : BOOL; (*Back Of Last Bag*)
		NewPatternOneShot : BOOL; (*New Pattern One Shot*)
		EndOfRun : BOOL; (*End Of Run EOR*)
	END_STRUCT;
END_TYPE

(*********************************************************************************
appControlCmd_typ
*********************************************************************************)

TYPE
	appMachineStatus_typ : 	STRUCT  (*Application Control Commands*)
		machine_running : BOOL; (*Machine Running AUTO*)
	END_STRUCT;
END_TYPE

(*********************************************************************************
appControlCmd_typ
*********************************************************************************)

TYPE
	appControlCmd_typ : 	STRUCT  (*Application Control Commands*)
		acknowledge_btn : BOOL; (*Acknowledge Button*)
		machine_start : BOOL; (*Machine Start*)
		machine_stop : BOOL; (*Machine Stop*)
		guard_eye_reset : BOOL; (*Guard Eye Reset PB5 ???*)
		pallet_discharge_selector_switch : BOOL; (*Pallet Discharge Selector Switch???*)
	END_STRUCT;
	appPalleteCfg_typ : 	STRUCT  (*Application Control Commands*)
		palleteSizeIdx : UDINT; (*Acknowledge Button*)
		layerCount : UDINT; (*Machine Start*)
		layerPatternIdx : ARRAY[0..15]OF UDINT; (*Machine Start*)
		layerUseTierSheet : ARRAY[0..15]OF UDINT; (*Machine Start*)
		layerOption1 : ARRAY[0..15]OF UDINT; (*Machine Start*)
	END_STRUCT;
	appPalleteCtrl_typ : 	STRUCT  (*Application Control Commands*)
		layerVisibility : ARRAY[0..15]OF USINT; (*Acknowledge Button*)
		layerCount : UDINT; (*Machine Start*)
	END_STRUCT;
END_TYPE

(*========================================================*)
(*Pallete configuration (recipe) structures*)
(*========================================================*)

TYPE
	palleteCfgSettings_typ : 	STRUCT  (*Pallete configuration (recipe) settings*)
		testTimer1 : REAL;
		timers : appCfgTimers_typ;
		vfd : ARRAY[0..APP_VFD_IDXLAST]OF cfgMachineVFDs_typ;
	END_STRUCT;
	palleteCfgLayerSettings_typ : 	STRUCT  (*Pallete configuration (recipe) settings*)
		layerFilename : STRING[31]; (*filename of the layer program to use*)
		insertTearSheet : UDINT; (*feature: insert tear sheet*)
		layerFeature1 : UDINT; (*feature: tbd*)
		sameAsOtherLayer : UDINT; (*0-not used at all; 1-use settings/configuration from the other layer (i.e. layerFilename not used, local values here not used);2-use layer settings*)
		otherLayerIdx : UDINT; (*if useOtherLayer=1, this is the index of the layer to use (0..maxLayerIdx)*)
	END_STRUCT;
	palleteCfgDimensions_typ : 	STRUCT  (*Pallete configuration (recipe) dimensions*)
		caseWidth : REAL;
		caseLength : REAL;
		caseHeight : REAL;
		palleteHeight : REAL;
		palleteWidth : REAL;
		palleteLength : REAL;
		palleteSizeHmiIdx : UDINT;
	END_STRUCT;
	palleteCfgCmdsTxt_typ : 	STRUCT  (*Pallete configuration program single instruction*)
		colorIdx : UDINT; (*0-none;1-case; 2-case +90 deg; 3-case -90 deg; 4-case 180 deg; *)
		cmdTxt : STRING[31];
	END_STRUCT;
	palleteCfgCmds_typ : 	STRUCT  (*Pallete configuration program single instruction*)
		cmdCase : USINT; (*0-none;1-case; 2-case +90 deg; 3-case -90 deg; 4-case 180 deg; *)
		cmdBlade : USINT; (*0-none, 1-bladeStop1; 2-bladeStop2, etc*)
		cmdFeature : USINT; (*0-none; 1-tbd*)
		cmdExtra : USINT; (*0-none; 1-tbd*)
	END_STRUCT;
	palleteCfgRowTxt_typ : 	STRUCT  (*Pallete row configuration (recipe) structure - collection of single instructions*)
		palCfgCmdsTxt : ARRAY[0..11]OF palleteCfgCmdsTxt_typ;
	END_STRUCT;
	palleteCfgRow_typ : 	STRUCT  (*Pallete row configuration (recipe) structure - collection of single instructions*)
		palCfgCmds : ARRAY[0..11]OF palleteCfgCmds_typ;
	END_STRUCT;
	palleteCfgLayerTxt_typ : 	STRUCT  (*Pallete layer configuration (recipe) structure - collection of rows*)
		layerFilename : STRING[31];
		layerDescription : STRING[31];
		curIdxEditorCell : UDINT;
		curIdxEditorCellOld : UDINT;
		curIdxRow : UDINT;
		curIdxCmd : UDINT;
		curCmdTxt : STRING[31];
		cmdIdxBlade : USINT;
		cmdIdxCase : USINT;
		cmdEntryCompletion : USINT;
		palCfgRowsTxt : ARRAY[0..11]OF palleteCfgRowTxt_typ;
	END_STRUCT;
	palleteCfgLayer_typ : 	STRUCT  (*Pallete layer configuration (recipe) structure - collection of rows*)
		layerFilename : STRING[31];
		layerDescription : STRING[31];
		palCfgRows : ARRAY[0..11]OF palleteCfgRow_typ;
	END_STRUCT;
	palleteCfg_typ : 	STRUCT  (*Pallete configuration (recipe) structure - collection of layers*)
		palFilename : STRING[31];
		palDescription : STRING[31];
		palActiveLayers : UDINT;
		palSettings : palleteCfgSettings_typ;
		palDimensions : palleteCfgDimensions_typ;
		palLayerSettings : ARRAY[0..11]OF palleteCfgLayerSettings_typ;
		magicNumber : UDINT;
	END_STRUCT;
END_TYPE

(*========================================================*)
(*Pallete program control structures*)
(*========================================================*)

TYPE
	palleteCtrlProcessor_typ : 	STRUCT  (*Pallete control processor data*)
		ssmInfeed : bgSSM_typ;
		ssmLayer : bgSSM_typ; (*state machine - layer forming*)
		ssmElevator : bgSSM_typ; (*state machine - elevator control*)
		ssmPallete : bgSSM_typ; (*state machine - pallete infeed / outfeed*)
		cmdIdx : UDINT; (*Current command index (from the current row)*)
		rowIdx : UDINT; (*Current row index (from the current layer)*)
		layerIdx : UDINT; (*Current layer index (from the collection of pallete layers)*)
		oPalleteRecipeIsValid : UDINT; (*Output: 1-loaded pallete recipe program is valid and it may run; 0-load pallete recipe program is not valid *)
		oRowIdxDN : USINT;
		oLayerIdxDN : USINT;
		oPalletStart : BOOL;
		oRowDN : BOOL; (*Output: current row execution is complete*)
		oLayerDN : BOOL; (*Output: current layer execution is complete*)
		oPalletDN : BOOL; (*Output: current case execution is complete*)
		oCaseDN : BOOL;
		oCurrentCases : UDINT; (*Current  number of cases processed for the entire pallet*)
		oTargetCases : UDINT; (*Target number of cases for the current row*)
		oTargetRows : UDINT; (*Targe number of rows for the current layer*)
		oTargetLayers : UDINT; (*Target number of layers for the pallet*)
		oTargetPalletCases : UDINT; (*Total number of target cases for the pallet*)
		iPause : UDINT; (*External input: pause execution*)
		iContinue : UDINT; (*External input: continue / resume execution*)
		iReset : UDINT; (*External input: reset execution*)
		iSet : UDINT; (*External input: set state of the processor execution*)
		iSetParamRow : UDINT; (*External input: parameter for the set state -  execution row*)
		iSetParamLayer : UDINT; (*External input: parameter for the set state - execution layer*)
		cmdBreakpoint : UDINT;
	END_STRUCT;
	palleteCtrlCmds_typ : 	STRUCT
		cmdActive : SINT; (*0-none;1-case; 2-case +90 deg; 3-case -90 deg; 4-case 180 deg; *)
		cmdVisible : SINT; (*0-none, 1-bladeStop1; 2-bladeStop2, etc*)
		cmdBreakpoint : SINT; (*0-none; 1-tbd*)
		cmdExtra : SINT; (*0-none; 1-tbd*)
	END_STRUCT;
	palleteCtrlRow_typ : 	STRUCT  (*Pallete row configuration (recipe) structure - collection of single instructions*)
		palCtrlCmds : ARRAY[0..11]OF palleteCtrlCmds_typ;
	END_STRUCT;
	palleteCtrlLayer_typ : 	STRUCT  (*Pallete layer configuration (recipe) structure - collection of rows*)
		btnAssignLayerFilename : USINT;
		btnDeleteLayerFilename : USINT;
		layerVisible : USINT;
		tearSheetOptionVisible : USINT;
		option1Visible : USINT;
		palCtrlRows : ARRAY[0..11]OF palleteCtrlRow_typ;
	END_STRUCT;
	palleteCtrl_typ : 	STRUCT  (*Pallete runtime control structure*)
		palCfg : palleteCfg_typ; (*Active pallete configuration - loaded/saved to/from a pallete recipe file*)
		palCfgLayers : ARRAY[0..11]OF palleteCfgLayer_typ; (*Active layer configuration for the active pallete - each layer structure loaded from an appropriate layer file (speficied in the pallet structure)*)
		ctrlLayers : ARRAY[0..11]OF palleteCtrlLayer_typ; (*Layer control structures used during runtime to control / operate layer loading*)
		ctrlProc : palleteCtrlProcessor_typ; (*Pallete building processor control structure*)
	END_STRUCT;
END_TYPE

(*========================================================*)
(*Animation stuff*)
(*========================================================*)

TYPE
	appHmiFileHandling_typ : 	STRUCT
		iBtnLoadL1Preview : USINT;
		iBtnLoadL2Preview : USINT;
		iBtnLoad : USINT;
		iBtnSave : USINT;
		iBtnNew : USINT;
		fileHandlerState : UDINT;
		fileHandlerTimer : TON;
	END_STRUCT;
END_TYPE

(*========================================================*)
(*Animation stuff*)
(*========================================================*)

TYPE
	appControlAnimationRow_typ : 	STRUCT  (*Application Animation Control*)
		animationRow : ARRAY[0..9]OF UDINT;
	END_STRUCT;
	appControlAnimation_typ : 	STRUCT  (*Application Animation Control*)
		tmrCase : TON;
		New_Member1 : USINT;
		New_Member : USINT;
		currentCase : UDINT;
		currentRow : UDINT;
		currentLayer : UDINT;
		visiCase : appControlAnimationRow_typ;
		visiRow : ARRAY[0..9]OF appControlAnimationRow_typ;
		visiLayer : ARRAY[0..9]OF appControlAnimationRow_typ;
	END_STRUCT;
END_TYPE
```

### MachineControl.var - Global variables
```iecst
(*Main Control Object*)
VAR
	gCtrl : macCtrl_typ := (0);
	gCtrlAnimation : appControlAnimation_typ := (0);
	dryCycleState : UDINT := 0;
	dryCycleStatePallete : UDINT := 0;
	animationState : UDINT := 0;
	gMsgRunning : STRING[63] := 'Palletizer 72';
	gMsgRunningCtrl : paiHmiMsgRunning_typ := (0);
END_VAR
(*==========================================================*)
VAR RETAIN
	gPallete : palleteCtrl_typ := (0);
END_VAR
VAR
	gLayer_L0 : palleteCfgLayer_typ := (0);
	gLayer_L1 : palleteCfgLayer_typ := (0);
	gLayerEditor : palleteCfgLayer_typ := (0);
	gLayerEditorTxt : palleteCfgLayerTxt_typ := (0);
END_VAR
(*Application specific recipe file handling*)
VAR
	gPalleteFileHandler : appHmiFileHandling_typ := (0);
	gLayerFileHandler : appHmiFileHandling_typ := (0);
	gLayer_L0_L1_FileHandler : appHmiFileHandling_typ := (0);
END_VAR
VAR RETAIN
	gStats : macCtrlStats_typ := (0);
END_VAR
```

### Program Logical/MachineControl/machCtrl (ANSIC) - app Machine Control

#### Cyclic.c - Cyclic code
```c
#include <bur/plctypes.h>

#ifdef _DEFAULT_INCLUDES
	#include <AsDefault.h>
#endif

#include "../../paiComponents/paiHmi/paiHmiMsgScrolling.h"

#if 1
#include <../../paiComponents/bglib/bgPVLogger3.c>
#define LOG_ENTRY_COUNT 30	//max number of log entries
#define LOG_ENTRY_LENGTH  200//max length of individual log message. Longer msg are truncated
_LOCAL STRING log[LOG_ENTRY_COUNT][LOG_ENTRY_LENGTH]; //log output visible from Automation Studio!
//static bgPVLogger_typ lgr;	//PV logger object
#else
#define DBG(format, args...) ;
#define DBGINIT(args...) ;
#endif

/*
###############################################################################
Alarms & Messages
###############################################################################
*/
static void machCtrlAlarms()
{
	int ii;
	//auxiliary service - scan all alarms
	gAlarms.oIsAlarmActive = 0;
	gAlarms.oIsAlarmActiveCount = 0;
	gAlarms.oIsAlarmNotAckCount = 0;
	for(ii=0; ii<=APP_ALARM_LASTTOCHECK; ii++){
		if(gAlarms.alarmActive[ii]){
			gAlarms.oIsAlarmActiveCount++;
			gAlarms.oIsAlarmActive = 1;
		}
	}
	gAlarms.oIsAlarmNotAck = 0;
	for(ii=0; ii<=APP_ALARM_LASTTOCHECK; ii++){
		if(gAlarms.alarmAck[ii]){
			gAlarms.oIsAlarmNotAckCount++;
			gAlarms.oIsAlarmNotAck = 1;
		}
	}

	for(ii=0; ii<=APP_ALARM_LASTTOCHECK; ii++){
		if((gAlarms.alarmActive[ii] || gAlarms.alarmAck[ii]) && (ii != APP_ALARM_AIRPRESSURE) ){
			gAlarmsFiltered.alarmActive[ii] = 1;
		}else{
			gAlarmsFiltered.alarmActive[ii] = 0;
		}
	}

	if((gAlarms.oIsAlarmNotAckCount <= 1) && (gAlarms.alarmActive[APP_ALARM_AIRPRESSURE])){
		gAlarmsFiltered.alarmActive[APP_ALARM_AIRPRESSURE] = 1;
	}

	//messages (yellow information box) are enabled only if alarms are not active
	//gMsgScroll.iEnable = gAlarms.oIsAlarmActive ? 0 : 1;
	gMsgScroll.iEnable = 1;
	paiHmiMsgScrollingCyclic(&gMsgScroll);

	//keep looking for a missing module alarm
	gAlarms.alarmActive[APP_ALARM_HWMODULE] = 0;
	for(ii=1; ii<APP_HWMODULE_IDXLAST; ii++){
		if( !gHWModules[ii].ModuleOk ){
			gAlarms.alarmActive[APP_ALARM_HWMODULE] = 1;
		}
	}

}
/*
###############################################################################
Init, Cyclic, Exit
###############################################################################
*/
void _INIT machCtrlInit(void)
{
	/* TODO: Add code here */
	DBGINIT(lgr, log, LOG_ENTRY_COUNT, LOG_ENTRY_LENGTH);

	gMachineIO.din.AuxVFDsOk = 0;
	gHWModules[0].ModuleOk = 0;
	gMachineVFD[0].appID = 0;
	gMachineVFD[6].appID = 6;//USED DON'T CHANGED IT!!!

	brsstrcpy((UDINT)gProjectInfo.ProjectComments, (UDINT)"gb comment");

	//Message scrolling support - init
	gMsgScroll.iEnable = 1;
	paiHmiMsgScrollingInit(&gMsgScroll, (UDINT)&gMessages.msgActive[0], APP_MSG_LAST + 1, 2000);

}

void _CYCLIC machCtrlCyclic(void)
{
	machCtrlAlarms();
}
```

- paiHmiMsgScrolling.c (reference to Logical/paiComponents/paiHmi/paiHmiMsgScrolling.c)

- bgstring.c (reference to Logical/paiComponents/bglib/bgstring.c)

- Program Logical/MachineControl/vfdControl (ANSIC) - app VFD Control (no source held here)

### Program Logical/MachineControl/palProc (ANSIC) - app Pallet Processor

- bgstring.c (reference to Logical/paiComponents/bglib/bgstring.c)

### Program Logical/MachineControl/appDraw (ANSIC) - app Drawing
